aff1Al[0  , 0] := 1.00000E+01; aff1Al[0  , 1] := -9.84199E+00;
aff1Al[1  , 0] := 1.99800E+01; aff1Al[1  , 1] := -1.00077E+01;
aff1Al[2  , 0] := 2.99600E+01; aff1Al[2  , 1] := -1.02348E+01;
aff1Al[3  , 0] := 3.99400E+01; aff1Al[3  , 1] := -1.05422E+01;
aff1Al[4  , 0] := 4.99200E+01; aff1Al[4  , 1] := -1.10354E+01;
aff1Al[5  , 0] := 5.99000E+01; aff1Al[5  , 1] := -1.19198E+01;
aff1Al[6  , 0] := 6.98800E+01; aff1Al[6  , 1] := -1.41453E+01;
aff1Al[7  , 0] := 7.98600E+01; aff1Al[7  , 1] := -1.44478E+01;
aff1Al[8  , 0] := 8.98400E+01; aff1Al[8  , 1] := -1.31089E+01;
aff1Al[9  , 0] := 9.98200E+01; aff1Al[9  , 1] := -1.16796E+01;
aff1Al[10 , 0] := 1.09800E+02; aff1Al[10 , 1] := -1.03556E+01;
aff1Al[11 , 0] := 1.19780E+02; aff1Al[11 , 1] := -9.31746E+00;
aff1Al[12 , 0] := 1.29760E+02; aff1Al[12 , 1] := -7.63743E+00;
aff1Al[13 , 0] := 1.39740E+02; aff1Al[13 , 1] := -6.42389E+00;
aff1Al[14 , 0] := 1.49720E+02; aff1Al[14 , 1] := -5.44289E+00;
aff1Al[15 , 0] := 1.59700E+02; aff1Al[15 , 1] := -4.64208E+00;
aff1Al[16 , 0] := 1.69680E+02; aff1Al[16 , 1] := -3.98698E+00;
aff1Al[17 , 0] := 1.79660E+02; aff1Al[17 , 1] := -3.45000E+00;
aff1Al[18 , 0] := 1.89640E+02; aff1Al[18 , 1] := -3.00860E+00;
aff1Al[19 , 0] := 1.99620E+02; aff1Al[19 , 1] := -2.64455E+00;
aff1Al[20 , 0] := 2.09600E+02; aff1Al[20 , 1] := -2.34326E+00;
aff1Al[21 , 0] := 2.19580E+02; aff1Al[21 , 1] := -2.09321E+00;
aff1Al[22 , 0] := 2.29560E+02; aff1Al[22 , 1] := -1.88468E+00;
aff1Al[23 , 0] := 2.39540E+02; aff1Al[23 , 1] := -1.71030E+00;
aff1Al[24 , 0] := 2.49520E+02; aff1Al[24 , 1] := -1.56408E+00;
aff1Al[25 , 0] := 2.59500E+02; aff1Al[25 , 1] := -1.44116E+00;
aff1Al[26 , 0] := 2.69480E+02; aff1Al[26 , 1] := -1.33759E+00;
aff1Al[27 , 0] := 2.79460E+02; aff1Al[27 , 1] := -1.25018E+00;
aff1Al[28 , 0] := 2.89440E+02; aff1Al[28 , 1] := -1.17627E+00;
aff1Al[29 , 0] := 2.99420E+02; aff1Al[29 , 1] := -1.11369E+00;
aff1Al[30 , 0] := 3.09400E+02; aff1Al[30 , 1] := -1.06082E+00;
aff1Al[31 , 0] := 3.19380E+02; aff1Al[31 , 1] := -1.01635E+00;
aff1Al[32 , 0] := 3.29360E+02; aff1Al[32 , 1] := -9.79160E-01;
aff1Al[33 , 0] := 3.39340E+02; aff1Al[33 , 1] := -9.48230E-01;
aff1Al[34 , 0] := 3.49320E+02; aff1Al[34 , 1] := -9.22697E-01;
aff1Al[35 , 0] := 3.59300E+02; aff1Al[35 , 1] := -9.02016E-01;
aff1Al[36 , 0] := 3.69280E+02; aff1Al[36 , 1] := -8.85231E-01;
aff1Al[37 , 0] := 3.79260E+02; aff1Al[37 , 1] := -8.71960E-01;
aff1Al[38 , 0] := 3.89240E+02; aff1Al[38 , 1] := -8.61750E-01;
aff1Al[39 , 0] := 3.99220E+02; aff1Al[39 , 1] := -8.54204E-01;
aff1Al[40 , 0] := 4.09200E+02; aff1Al[40 , 1] := -8.48983E-01;
aff1Al[41 , 0] := 4.19180E+02; aff1Al[41 , 1] := -8.45791E-01;
aff1Al[42 , 0] := 4.29160E+02; aff1Al[42 , 1] := -8.44376E-01;
aff1Al[43 , 0] := 4.39140E+02; aff1Al[43 , 1] := -8.44514E-01;
aff1Al[44 , 0] := 4.49120E+02; aff1Al[44 , 1] := -8.46014E-01;
aff1Al[45 , 0] := 4.59100E+02; aff1Al[45 , 1] := -8.48707E-01;
aff1Al[46 , 0] := 4.69080E+02; aff1Al[46 , 1] := -8.52446E-01;
aff1Al[47 , 0] := 4.79060E+02; aff1Al[47 , 1] := -8.57102E-01;
aff1Al[48 , 0] := 4.89040E+02; aff1Al[48 , 1] := -8.62576E-01;
aff1Al[49 , 0] := 4.99020E+02; aff1Al[49 , 1] := -8.68781E-01;
aff1Al[50 , 0] := 5.09000E+02; aff1Al[50 , 1] := -8.75639E-01;
aff1Al[51 , 0] := 5.18980E+02; aff1Al[51 , 1] := -8.83079E-01;
aff1Al[52 , 0] := 5.28960E+02; aff1Al[52 , 1] := -8.91040E-01;
aff1Al[53 , 0] := 5.38940E+02; aff1Al[53 , 1] := -8.99464E-01;
aff1Al[54 , 0] := 5.48920E+02; aff1Al[54 , 1] := -9.08301E-01;
aff1Al[55 , 0] := 5.58900E+02; aff1Al[55 , 1] := -9.17508E-01;
aff1Al[56 , 0] := 5.68880E+02; aff1Al[56 , 1] := -9.27045E-01;
aff1Al[57 , 0] := 5.78860E+02; aff1Al[57 , 1] := -9.36877E-01;
aff1Al[58 , 0] := 5.88840E+02; aff1Al[58 , 1] := -9.46974E-01;
aff1Al[59 , 0] := 5.98820E+02; aff1Al[59 , 1] := -9.57307E-01;
aff1Al[60 , 0] := 6.08800E+02; aff1Al[60 , 1] := -9.67854E-01;
aff1Al[61 , 0] := 6.18780E+02; aff1Al[61 , 1] := -9.78593E-01;
aff1Al[62 , 0] := 6.28760E+02; aff1Al[62 , 1] := -9.89506E-01;
aff1Al[63 , 0] := 6.38740E+02; aff1Al[63 , 1] := -1.00058E+00;
aff1Al[64 , 0] := 6.48720E+02; aff1Al[64 , 1] := -1.01179E+00;
aff1Al[65 , 0] := 6.58700E+02; aff1Al[65 , 1] := -1.02313E+00;
aff1Al[66 , 0] := 6.68680E+02; aff1Al[66 , 1] := -1.03460E+00;
aff1Al[67 , 0] := 6.78660E+02; aff1Al[67 , 1] := -1.04617E+00;
aff1Al[68 , 0] := 6.88640E+02; aff1Al[68 , 1] := -1.05785E+00;
aff1Al[69 , 0] := 6.98620E+02; aff1Al[69 , 1] := -1.06963E+00;
aff1Al[70 , 0] := 7.08600E+02; aff1Al[70 , 1] := -1.08150E+00;
aff1Al[71 , 0] := 7.18580E+02; aff1Al[71 , 1] := -1.09346E+00;
aff1Al[72 , 0] := 7.28560E+02; aff1Al[72 , 1] := -1.10551E+00;
aff1Al[73 , 0] := 7.38540E+02; aff1Al[73 , 1] := -1.11763E+00;
aff1Al[74 , 0] := 7.48520E+02; aff1Al[74 , 1] := -1.12984E+00;
aff1Al[75 , 0] := 7.58500E+02; aff1Al[75 , 1] := -1.14213E+00;
aff1Al[76 , 0] := 7.68480E+02; aff1Al[76 , 1] := -1.15450E+00;
aff1Al[77 , 0] := 7.78460E+02; aff1Al[77 , 1] := -1.16695E+00;
aff1Al[78 , 0] := 7.88440E+02; aff1Al[78 , 1] := -1.17949E+00;
aff1Al[79 , 0] := 7.98420E+02; aff1Al[79 , 1] := -1.19211E+00;
aff1Al[80 , 0] := 8.08400E+02; aff1Al[80 , 1] := -1.20481E+00;
aff1Al[81 , 0] := 8.18380E+02; aff1Al[81 , 1] := -1.21760E+00;
aff1Al[82 , 0] := 8.28360E+02; aff1Al[82 , 1] := -1.23049E+00;
aff1Al[83 , 0] := 8.38340E+02; aff1Al[83 , 1] := -1.24347E+00;
aff1Al[84 , 0] := 8.48320E+02; aff1Al[84 , 1] := -1.25655E+00;
aff1Al[85 , 0] := 8.58300E+02; aff1Al[85 , 1] := -1.26974E+00;
aff1Al[86 , 0] := 8.68280E+02; aff1Al[86 , 1] := -1.28303E+00;
aff1Al[87 , 0] := 8.78260E+02; aff1Al[87 , 1] := -1.29644E+00;
aff1Al[88 , 0] := 8.88240E+02; aff1Al[88 , 1] := -1.30997E+00;
aff1Al[89 , 0] := 8.98220E+02; aff1Al[89 , 1] := -1.32363E+00;
aff1Al[90 , 0] := 9.08200E+02; aff1Al[90 , 1] := -1.33742E+00;
aff1Al[91 , 0] := 9.18180E+02; aff1Al[91 , 1] := -1.35136E+00;
aff1Al[92 , 0] := 9.28160E+02; aff1Al[92 , 1] := -1.36544E+00;
aff1Al[93 , 0] := 9.38140E+02; aff1Al[93 , 1] := -1.37968E+00;
aff1Al[94 , 0] := 9.48120E+02; aff1Al[94 , 1] := -1.39408E+00;
aff1Al[95 , 0] := 9.58100E+02; aff1Al[95 , 1] := -1.40865E+00;
aff1Al[96 , 0] := 9.68080E+02; aff1Al[96 , 1] := -1.42341E+00;
aff1Al[97 , 0] := 9.78060E+02; aff1Al[97 , 1] := -1.43836E+00;
aff1Al[98 , 0] := 9.88040E+02; aff1Al[98 , 1] := -1.45353E+00;
aff1Al[99 , 0] := 9.98020E+02; aff1Al[99 , 1] := -1.46877E+00;
aff1Al[100, 0] := 1.00800E+03; aff1Al[100, 1] := -1.47677E+00;
aff1Al[101, 0] := 1.01798E+03; aff1Al[101, 1] := -1.49037E+00;
aff1Al[102, 0] := 1.02796E+03; aff1Al[102, 1] := -1.50547E+00;
aff1Al[103, 0] := 1.03794E+03; aff1Al[103, 1] := -1.52135E+00;
aff1Al[104, 0] := 1.04792E+03; aff1Al[104, 1] := -1.53779E+00;
aff1Al[105, 0] := 1.05790E+03; aff1Al[105, 1] := -1.55471E+00;
aff1Al[106, 0] := 1.06788E+03; aff1Al[106, 1] := -1.57209E+00;
aff1Al[107, 0] := 1.07786E+03; aff1Al[107, 1] := -1.58990E+00;
aff1Al[108, 0] := 1.08784E+03; aff1Al[108, 1] := -1.60814E+00;
aff1Al[109, 0] := 1.09782E+03; aff1Al[109, 1] := -1.62683E+00;
aff1Al[110, 0] := 1.10780E+03; aff1Al[110, 1] := -1.64597E+00;
aff1Al[111, 0] := 1.11778E+03; aff1Al[111, 1] := -1.66557E+00;
aff1Al[112, 0] := 1.12776E+03; aff1Al[112, 1] := -1.68565E+00;
aff1Al[113, 0] := 1.13774E+03; aff1Al[113, 1] := -1.70624E+00;
aff1Al[114, 0] := 1.14772E+03; aff1Al[114, 1] := -1.72735E+00;
aff1Al[115, 0] := 1.15770E+03; aff1Al[115, 1] := -1.74901E+00;
aff1Al[116, 0] := 1.16768E+03; aff1Al[116, 1] := -1.77126E+00;
aff1Al[117, 0] := 1.17766E+03; aff1Al[117, 1] := -1.79411E+00;
aff1Al[118, 0] := 1.18764E+03; aff1Al[118, 1] := -1.81762E+00;
aff1Al[119, 0] := 1.19762E+03; aff1Al[119, 1] := -1.84181E+00;
aff1Al[120, 0] := 1.20760E+03; aff1Al[120, 1] := -1.86674E+00;
aff1Al[121, 0] := 1.21758E+03; aff1Al[121, 1] := -1.89244E+00;
aff1Al[122, 0] := 1.22756E+03; aff1Al[122, 1] := -1.91897E+00;
aff1Al[123, 0] := 1.23754E+03; aff1Al[123, 1] := -1.94639E+00;
aff1Al[124, 0] := 1.24752E+03; aff1Al[124, 1] := -1.97475E+00;
aff1Al[125, 0] := 1.25750E+03; aff1Al[125, 1] := -2.00414E+00;
aff1Al[126, 0] := 1.26748E+03; aff1Al[126, 1] := -2.03461E+00;
aff1Al[127, 0] := 1.27746E+03; aff1Al[127, 1] := -2.06626E+00;
aff1Al[128, 0] := 1.28744E+03; aff1Al[128, 1] := -2.09918E+00;
aff1Al[129, 0] := 1.29742E+03; aff1Al[129, 1] := -2.13348E+00;
aff1Al[130, 0] := 1.30740E+03; aff1Al[130, 1] := -2.16927E+00;
aff1Al[131, 0] := 1.31738E+03; aff1Al[131, 1] := -2.20668E+00;
aff1Al[132, 0] := 1.32736E+03; aff1Al[132, 1] := -2.24586E+00;
aff1Al[133, 0] := 1.33734E+03; aff1Al[133, 1] := -2.28699E+00;
aff1Al[134, 0] := 1.34732E+03; aff1Al[134, 1] := -2.33024E+00;
aff1Al[135, 0] := 1.35730E+03; aff1Al[135, 1] := -2.37585E+00;
aff1Al[136, 0] := 1.36728E+03; aff1Al[136, 1] := -2.42407E+00;
aff1Al[137, 0] := 1.37726E+03; aff1Al[137, 1] := -2.47520E+00;
aff1Al[138, 0] := 1.38724E+03; aff1Al[138, 1] := -2.52958E+00;
aff1Al[139, 0] := 1.39722E+03; aff1Al[139, 1] := -2.58764E+00;
aff1Al[140, 0] := 1.40720E+03; aff1Al[140, 1] := -2.64987E+00;
aff1Al[141, 0] := 1.41718E+03; aff1Al[141, 1] := -2.71687E+00;
aff1Al[142, 0] := 1.42716E+03; aff1Al[142, 1] := -2.78934E+00;
aff1Al[143, 0] := 1.43714E+03; aff1Al[143, 1] := -2.86819E+00;
aff1Al[144, 0] := 1.44712E+03; aff1Al[144, 1] := -2.95455E+00;
aff1Al[145, 0] := 1.45710E+03; aff1Al[145, 1] := -3.04985E+00;
aff1Al[146, 0] := 1.46708E+03; aff1Al[146, 1] := -3.15601E+00;
aff1Al[147, 0] := 1.47706E+03; aff1Al[147, 1] := -3.27556E+00;
aff1Al[148, 0] := 1.48704E+03; aff1Al[148, 1] := -3.41203E+00;
aff1Al[149, 0] := 1.49702E+03; aff1Al[149, 1] := -3.57073E+00;
aff1Al[150, 0] := 1.50700E+03; aff1Al[150, 1] := -3.75998E+00;
aff1Al[151, 0] := 1.51698E+03; aff1Al[151, 1] := -3.99072E+00;
aff1Al[152, 0] := 1.52696E+03; aff1Al[152, 1] := -4.28999E+00;
aff1Al[153, 0] := 1.53694E+03; aff1Al[153, 1] := -4.69289E+00;
aff1Al[154, 0] := 1.54692E+03; aff1Al[154, 1] := -5.36933E+00;
aff1Al[155, 0] := 1.55690E+03; aff1Al[155, 1] := -7.18317E+00;
aff1Al[156, 0] := 1.56688E+03; aff1Al[156, 1] := -6.04049E+00;
aff1Al[157, 0] := 1.57686E+03; aff1Al[157, 1] := -4.98882E+00;
aff1Al[158, 0] := 1.58684E+03; aff1Al[158, 1] := -4.41253E+00;
aff1Al[159, 0] := 1.59682E+03; aff1Al[159, 1] := -4.02524E+00;
aff1Al[160, 0] := 1.60680E+03; aff1Al[160, 1] := -3.71526E+00;
aff1Al[161, 0] := 1.61678E+03; aff1Al[161, 1] := -3.45829E+00;
aff1Al[162, 0] := 1.62676E+03; aff1Al[162, 1] := -3.23561E+00;
aff1Al[163, 0] := 1.63674E+03; aff1Al[163, 1] := -3.03403E+00;
aff1Al[164, 0] := 1.64672E+03; aff1Al[164, 1] := -2.85340E+00;
aff1Al[165, 0] := 1.65670E+03; aff1Al[165, 1] := -2.69189E+00;
aff1Al[166, 0] := 1.66668E+03; aff1Al[166, 1] := -2.54596E+00;
aff1Al[167, 0] := 1.67666E+03; aff1Al[167, 1] := -2.41278E+00;
aff1Al[168, 0] := 1.68664E+03; aff1Al[168, 1] := -2.28993E+00;
aff1Al[169, 0] := 1.69662E+03; aff1Al[169, 1] := -2.17603E+00;
aff1Al[170, 0] := 1.70660E+03; aff1Al[170, 1] := -2.06993E+00;
aff1Al[171, 0] := 1.71658E+03; aff1Al[171, 1] := -1.97068E+00;
aff1Al[172, 0] := 1.72656E+03; aff1Al[172, 1] := -1.87755E+00;
aff1Al[173, 0] := 1.73654E+03; aff1Al[173, 1] := -1.78991E+00;
aff1Al[174, 0] := 1.74652E+03; aff1Al[174, 1] := -1.70725E+00;
aff1Al[175, 0] := 1.75650E+03; aff1Al[175, 1] := -1.62914E+00;
aff1Al[176, 0] := 1.76648E+03; aff1Al[176, 1] := -1.55520E+00;
aff1Al[177, 0] := 1.77646E+03; aff1Al[177, 1] := -1.48511E+00;
aff1Al[178, 0] := 1.78644E+03; aff1Al[178, 1] := -1.41857E+00;
aff1Al[179, 0] := 1.79642E+03; aff1Al[179, 1] := -1.35535E+00;
aff1Al[180, 0] := 1.80640E+03; aff1Al[180, 1] := -1.29521E+00;
aff1Al[181, 0] := 1.81638E+03; aff1Al[181, 1] := -1.23796E+00;
aff1Al[182, 0] := 1.82636E+03; aff1Al[182, 1] := -1.18341E+00;
aff1Al[183, 0] := 1.83634E+03; aff1Al[183, 1] := -1.13142E+00;
aff1Al[184, 0] := 1.84632E+03; aff1Al[184, 1] := -1.08181E+00;
aff1Al[185, 0] := 1.85630E+03; aff1Al[185, 1] := -1.03447E+00;
aff1Al[186, 0] := 1.86628E+03; aff1Al[186, 1] := -9.89263E-01;
aff1Al[187, 0] := 1.87626E+03; aff1Al[187, 1] := -9.46076E-01;
aff1Al[188, 0] := 1.88624E+03; aff1Al[188, 1] := -9.04806E-01;
aff1Al[189, 0] := 1.89622E+03; aff1Al[189, 1] := -8.65352E-01;
aff1Al[190, 0] := 1.90620E+03; aff1Al[190, 1] := -8.27626E-01;
aff1Al[191, 0] := 1.91618E+03; aff1Al[191, 1] := -7.91542E-01;
aff1Al[192, 0] := 1.92616E+03; aff1Al[192, 1] := -7.57024E-01;
aff1Al[193, 0] := 1.93614E+03; aff1Al[193, 1] := -7.23998E-01;
aff1Al[194, 0] := 1.94612E+03; aff1Al[194, 1] := -6.92399E-01;
aff1Al[195, 0] := 1.95610E+03; aff1Al[195, 1] := -6.62165E-01;
aff1Al[196, 0] := 1.96608E+03; aff1Al[196, 1] := -6.33242E-01;
aff1Al[197, 0] := 1.97606E+03; aff1Al[197, 1] := -6.05580E-01;
aff1Al[198, 0] := 1.98604E+03; aff1Al[198, 1] := -5.79132E-01;
aff1Al[199, 0] := 1.99602E+03; aff1Al[199, 1] := -5.53864E-01;
aff1Al[200, 0] := 2.00600E+03; aff1Al[200, 1] := -5.29790E-01;
aff1Al[201, 0] := 2.01598E+03; aff1Al[201, 1] := -5.06864E-01;
aff1Al[202, 0] := 2.02596E+03; aff1Al[202, 1] := -4.84983E-01;
aff1Al[203, 0] := 2.03594E+03; aff1Al[203, 1] := -4.63991E-01;
aff1Al[204, 0] := 2.04592E+03; aff1Al[204, 1] := -4.43605E-01;
aff1Al[205, 0] := 2.05590E+03; aff1Al[205, 1] := -4.23670E-01;
aff1Al[206, 0] := 2.06588E+03; aff1Al[206, 1] := -4.04256E-01;
aff1Al[207, 0] := 2.07586E+03; aff1Al[207, 1] := -3.85410E-01;
aff1Al[208, 0] := 2.08584E+03; aff1Al[208, 1] := -3.67104E-01;
aff1Al[209, 0] := 2.09582E+03; aff1Al[209, 1] := -3.49316E-01;
aff1Al[210, 0] := 2.10580E+03; aff1Al[210, 1] := -3.32036E-01;
aff1Al[211, 0] := 2.11578E+03; aff1Al[211, 1] := -3.15248E-01;
aff1Al[212, 0] := 2.12576E+03; aff1Al[212, 1] := -2.98937E-01;
aff1Al[213, 0] := 2.13574E+03; aff1Al[213, 1] := -2.83087E-01;
aff1Al[214, 0] := 2.14572E+03; aff1Al[214, 1] := -2.67681E-01;
aff1Al[215, 0] := 2.15570E+03; aff1Al[215, 1] := -2.52704E-01;
aff1Al[216, 0] := 2.16568E+03; aff1Al[216, 1] := -2.38139E-01;
aff1Al[217, 0] := 2.17566E+03; aff1Al[217, 1] := -2.23973E-01;
aff1Al[218, 0] := 2.18564E+03; aff1Al[218, 1] := -2.10191E-01;
aff1Al[219, 0] := 2.19562E+03; aff1Al[219, 1] := -1.96778E-01;
aff1Al[220, 0] := 2.20560E+03; aff1Al[220, 1] := -1.83722E-01;
aff1Al[221, 0] := 2.21558E+03; aff1Al[221, 1] := -1.71010E-01;
aff1Al[222, 0] := 2.22556E+03; aff1Al[222, 1] := -1.58630E-01;
aff1Al[223, 0] := 2.23554E+03; aff1Al[223, 1] := -1.46573E-01;
aff1Al[224, 0] := 2.24552E+03; aff1Al[224, 1] := -1.34830E-01;
aff1Al[225, 0] := 2.25550E+03; aff1Al[225, 1] := -1.23388E-01;
aff1Al[226, 0] := 2.26548E+03; aff1Al[226, 1] := -1.12239E-01;
aff1Al[227, 0] := 2.27546E+03; aff1Al[227, 1] := -1.01370E-01;
aff1Al[228, 0] := 2.28544E+03; aff1Al[228, 1] := -9.07737E-02;
aff1Al[229, 0] := 2.29542E+03; aff1Al[229, 1] := -8.04398E-02;
aff1Al[230, 0] := 2.30540E+03; aff1Al[230, 1] := -7.03599E-02;
aff1Al[231, 0] := 2.31538E+03; aff1Al[231, 1] := -6.05256E-02;
aff1Al[232, 0] := 2.32536E+03; aff1Al[232, 1] := -5.09289E-02;
aff1Al[233, 0] := 2.33534E+03; aff1Al[233, 1] := -4.15622E-02;
aff1Al[234, 0] := 2.34532E+03; aff1Al[234, 1] := -3.24183E-02;
aff1Al[235, 0] := 2.35530E+03; aff1Al[235, 1] := -2.34900E-02;
aff1Al[236, 0] := 2.36528E+03; aff1Al[236, 1] := -1.47706E-02;
aff1Al[237, 0] := 2.37526E+03; aff1Al[237, 1] := -6.25378E-03;
aff1Al[238, 0] := 2.38524E+03; aff1Al[238, 1] := 2.06666E-03;
aff1Al[239, 0] := 2.39522E+03; aff1Al[239, 1] := 1.01966E-02;
aff1Al[240, 0] := 2.40520E+03; aff1Al[240, 1] := 1.81418E-02;
aff1Al[241, 0] := 2.41518E+03; aff1Al[241, 1] := 2.59075E-02;
aff1Al[242, 0] := 2.42516E+03; aff1Al[242, 1] := 3.34991E-02;
aff1Al[243, 0] := 2.43514E+03; aff1Al[243, 1] := 4.09215E-02;
aff1Al[244, 0] := 2.44512E+03; aff1Al[244, 1] := 4.81795E-02;
aff1Al[245, 0] := 2.45510E+03; aff1Al[245, 1] := 5.52777E-02;
aff1Al[246, 0] := 2.46508E+03; aff1Al[246, 1] := 6.22206E-02;
aff1Al[247, 0] := 2.47506E+03; aff1Al[247, 1] := 6.90126E-02;
aff1Al[248, 0] := 2.48504E+03; aff1Al[248, 1] := 7.56575E-02;
aff1Al[249, 0] := 2.49502E+03; aff1Al[249, 1] := 8.21595E-02;
aff1Al[250, 0] := 2.50500E+03; aff1Al[250, 1] := 8.85222E-02;
aff1Al[251, 0] := 2.51498E+03; aff1Al[251, 1] := 9.47495E-02;
aff1Al[252, 0] := 2.52496E+03; aff1Al[252, 1] := 1.00845E-01;
aff1Al[253, 0] := 2.53494E+03; aff1Al[253, 1] := 1.06812E-01;
aff1Al[254, 0] := 2.54492E+03; aff1Al[254, 1] := 1.12653E-01;
aff1Al[255, 0] := 2.55490E+03; aff1Al[255, 1] := 1.18373E-01;
aff1Al[256, 0] := 2.56488E+03; aff1Al[256, 1] := 1.23973E-01;
aff1Al[257, 0] := 2.57486E+03; aff1Al[257, 1] := 1.29458E-01;
aff1Al[258, 0] := 2.58484E+03; aff1Al[258, 1] := 1.34829E-01;
aff1Al[259, 0] := 2.59482E+03; aff1Al[259, 1] := 1.40090E-01;
aff1Al[260, 0] := 2.60480E+03; aff1Al[260, 1] := 1.45244E-01;
aff1Al[261, 0] := 2.61478E+03; aff1Al[261, 1] := 1.50292E-01;
aff1Al[262, 0] := 2.62476E+03; aff1Al[262, 1] := 1.55239E-01;
aff1Al[263, 0] := 2.63474E+03; aff1Al[263, 1] := 1.60086E-01;
aff1Al[264, 0] := 2.64472E+03; aff1Al[264, 1] := 1.64833E-01;
aff1Al[265, 0] := 2.65470E+03; aff1Al[265, 1] := 1.69484E-01;
aff1Al[266, 0] := 2.66468E+03; aff1Al[266, 1] := 1.74040E-01;
aff1Al[267, 0] := 2.67466E+03; aff1Al[267, 1] := 1.78507E-01;
aff1Al[268, 0] := 2.68464E+03; aff1Al[268, 1] := 1.82888E-01;
aff1Al[269, 0] := 2.69462E+03; aff1Al[269, 1] := 1.87183E-01;
aff1Al[270, 0] := 2.70460E+03; aff1Al[270, 1] := 1.91394E-01;
aff1Al[271, 0] := 2.71458E+03; aff1Al[271, 1] := 1.95522E-01;
aff1Al[272, 0] := 2.72456E+03; aff1Al[272, 1] := 1.99569E-01;
aff1Al[273, 0] := 2.73454E+03; aff1Al[273, 1] := 2.03537E-01;
aff1Al[274, 0] := 2.74452E+03; aff1Al[274, 1] := 2.07429E-01;
aff1Al[275, 0] := 2.75450E+03; aff1Al[275, 1] := 2.11246E-01;
aff1Al[276, 0] := 2.76448E+03; aff1Al[276, 1] := 2.14990E-01;
aff1Al[277, 0] := 2.77446E+03; aff1Al[277, 1] := 2.18663E-01;
aff1Al[278, 0] := 2.78444E+03; aff1Al[278, 1] := 2.22266E-01;
aff1Al[279, 0] := 2.79442E+03; aff1Al[279, 1] := 2.25801E-01;
aff1Al[280, 0] := 2.80440E+03; aff1Al[280, 1] := 2.29270E-01;
aff1Al[281, 0] := 2.81438E+03; aff1Al[281, 1] := 2.32675E-01;
aff1Al[282, 0] := 2.82436E+03; aff1Al[282, 1] := 2.36016E-01;
aff1Al[283, 0] := 2.83434E+03; aff1Al[283, 1] := 2.39297E-01;
aff1Al[284, 0] := 2.84432E+03; aff1Al[284, 1] := 2.42518E-01;
aff1Al[285, 0] := 2.85430E+03; aff1Al[285, 1] := 2.45681E-01;
aff1Al[286, 0] := 2.86428E+03; aff1Al[286, 1] := 2.48789E-01;
aff1Al[287, 0] := 2.87426E+03; aff1Al[287, 1] := 2.51841E-01;
aff1Al[288, 0] := 2.88424E+03; aff1Al[288, 1] := 2.54841E-01;
aff1Al[289, 0] := 2.89422E+03; aff1Al[289, 1] := 2.57789E-01;
aff1Al[290, 0] := 2.90420E+03; aff1Al[290, 1] := 2.60688E-01;
aff1Al[291, 0] := 2.91418E+03; aff1Al[291, 1] := 2.63540E-01;
aff1Al[292, 0] := 2.92416E+03; aff1Al[292, 1] := 2.66349E-01;
aff1Al[293, 0] := 2.93414E+03; aff1Al[293, 1] := 2.69138E-01;
aff1Al[294, 0] := 2.94412E+03; aff1Al[294, 1] := 2.71862E-01;
aff1Al[295, 0] := 2.95410E+03; aff1Al[295, 1] := 2.74462E-01;
aff1Al[296, 0] := 2.96408E+03; aff1Al[296, 1] := 2.76910E-01;
aff1Al[297, 0] := 2.97406E+03; aff1Al[297, 1] := 2.79499E-01;
aff1Al[298, 0] := 2.98404E+03; aff1Al[298, 1] := 2.82539E-01;
aff1Al[299, 0] := 2.99402E+03; aff1Al[299, 1] := 2.86146E-01;
aff1Al[300, 0] := 3.00400E+03; aff1Al[300, 1] := 2.89853E-01;
aff1Al[301, 0] := 3.01398E+03; aff1Al[301, 1] := 2.93173E-01;
aff1Al[302, 0] := 3.02396E+03; aff1Al[302, 1] := 2.95852E-01;
aff1Al[303, 0] := 3.03394E+03; aff1Al[303, 1] := 2.98120E-01;
aff1Al[304, 0] := 3.04392E+03; aff1Al[304, 1] := 3.00329E-01;
aff1Al[305, 0] := 3.05390E+03; aff1Al[305, 1] := 3.02814E-01;
aff1Al[306, 0] := 3.06388E+03; aff1Al[306, 1] := 3.04933E-01;
aff1Al[307, 0] := 3.07386E+03; aff1Al[307, 1] := 3.05880E-01;
aff1Al[308, 0] := 3.08384E+03; aff1Al[308, 1] := 3.05153E-01;
aff1Al[309, 0] := 3.09382E+03; aff1Al[309, 1] := 3.06508E-01;
aff1Al[310, 0] := 3.10380E+03; aff1Al[310, 1] := 3.13763E-01;
aff1Al[311, 0] := 3.11378E+03; aff1Al[311, 1] := 3.29581E-01;
aff1Al[312, 0] := 3.12376E+03; aff1Al[312, 1] := 3.48098E-01;
aff1Al[313, 0] := 3.13374E+03; aff1Al[313, 1] := 3.63012E-01;
aff1Al[314, 0] := 3.14372E+03; aff1Al[314, 1] := 3.69087E-01;
aff1Al[315, 0] := 3.15370E+03; aff1Al[315, 1] := 3.69334E-01;
aff1Al[316, 0] := 3.16368E+03; aff1Al[316, 1] := 3.67698E-01;
aff1Al[317, 0] := 3.17366E+03; aff1Al[317, 1] := 3.67875E-01;
aff1Al[318, 0] := 3.18364E+03; aff1Al[318, 1] := 3.69502E-01;
aff1Al[319, 0] := 3.19362E+03; aff1Al[319, 1] := 3.71637E-01;
aff1Al[320, 0] := 3.20360E+03; aff1Al[320, 1] := 3.73286E-01;
aff1Al[321, 0] := 3.21358E+03; aff1Al[321, 1] := 3.74565E-01;
aff1Al[322, 0] := 3.22356E+03; aff1Al[322, 1] := 3.75687E-01;
aff1Al[323, 0] := 3.23354E+03; aff1Al[323, 1] := 3.76814E-01;
aff1Al[324, 0] := 3.24352E+03; aff1Al[324, 1] := 3.77939E-01;
aff1Al[325, 0] := 3.25350E+03; aff1Al[325, 1] := 3.79018E-01;
aff1Al[326, 0] := 3.26348E+03; aff1Al[326, 1] := 3.80052E-01;
aff1Al[327, 0] := 3.27346E+03; aff1Al[327, 1] := 3.81042E-01;
aff1Al[328, 0] := 3.28344E+03; aff1Al[328, 1] := 3.81991E-01;
aff1Al[329, 0] := 3.29342E+03; aff1Al[329, 1] := 3.82900E-01;
aff1Al[330, 0] := 3.30340E+03; aff1Al[330, 1] := 3.83769E-01;
aff1Al[331, 0] := 3.31338E+03; aff1Al[331, 1] := 3.84601E-01;
aff1Al[332, 0] := 3.32336E+03; aff1Al[332, 1] := 3.85396E-01;
aff1Al[333, 0] := 3.33334E+03; aff1Al[333, 1] := 3.86155E-01;
aff1Al[334, 0] := 3.34332E+03; aff1Al[334, 1] := 3.86880E-01;
aff1Al[335, 0] := 3.35330E+03; aff1Al[335, 1] := 3.87572E-01;
aff1Al[336, 0] := 3.36328E+03; aff1Al[336, 1] := 3.88231E-01;
aff1Al[337, 0] := 3.37326E+03; aff1Al[337, 1] := 3.88859E-01;
aff1Al[338, 0] := 3.38324E+03; aff1Al[338, 1] := 3.89456E-01;
aff1Al[339, 0] := 3.39322E+03; aff1Al[339, 1] := 3.90023E-01;
aff1Al[340, 0] := 3.40320E+03; aff1Al[340, 1] := 3.90562E-01;
aff1Al[341, 0] := 3.41318E+03; aff1Al[341, 1] := 3.91072E-01;
aff1Al[342, 0] := 3.42316E+03; aff1Al[342, 1] := 3.91555E-01;
aff1Al[343, 0] := 3.43314E+03; aff1Al[343, 1] := 3.92012E-01;
aff1Al[344, 0] := 3.44312E+03; aff1Al[344, 1] := 3.92443E-01;
aff1Al[345, 0] := 3.45310E+03; aff1Al[345, 1] := 3.92848E-01;
aff1Al[346, 0] := 3.46308E+03; aff1Al[346, 1] := 3.93229E-01;
aff1Al[347, 0] := 3.47306E+03; aff1Al[347, 1] := 3.93586E-01;
aff1Al[348, 0] := 3.48304E+03; aff1Al[348, 1] := 3.93920E-01;
aff1Al[349, 0] := 3.49302E+03; aff1Al[349, 1] := 3.94231E-01;
aff1Al[350, 0] := 3.50300E+03; aff1Al[350, 1] := 3.94520E-01;
aff1Al[351, 0] := 3.51298E+03; aff1Al[351, 1] := 3.94787E-01;
aff1Al[352, 0] := 3.52296E+03; aff1Al[352, 1] := 3.95033E-01;
aff1Al[353, 0] := 3.53294E+03; aff1Al[353, 1] := 3.95259E-01;
aff1Al[354, 0] := 3.54292E+03; aff1Al[354, 1] := 3.95465E-01;
aff1Al[355, 0] := 3.55290E+03; aff1Al[355, 1] := 3.95652E-01;
aff1Al[356, 0] := 3.56288E+03; aff1Al[356, 1] := 3.95819E-01;
aff1Al[357, 0] := 3.57286E+03; aff1Al[357, 1] := 3.95968E-01;
aff1Al[358, 0] := 3.58284E+03; aff1Al[358, 1] := 3.96099E-01;
aff1Al[359, 0] := 3.59282E+03; aff1Al[359, 1] := 3.96213E-01;
aff1Al[360, 0] := 3.60280E+03; aff1Al[360, 1] := 3.96309E-01;
aff1Al[361, 0] := 3.61278E+03; aff1Al[361, 1] := 3.96388E-01;
aff1Al[362, 0] := 3.62276E+03; aff1Al[362, 1] := 3.96451E-01;
aff1Al[363, 0] := 3.63274E+03; aff1Al[363, 1] := 3.96498E-01;
aff1Al[364, 0] := 3.64272E+03; aff1Al[364, 1] := 3.96529E-01;
aff1Al[365, 0] := 3.65270E+03; aff1Al[365, 1] := 3.96545E-01;
aff1Al[366, 0] := 3.66268E+03; aff1Al[366, 1] := 3.96547E-01;
aff1Al[367, 0] := 3.67266E+03; aff1Al[367, 1] := 3.96533E-01;
aff1Al[368, 0] := 3.68264E+03; aff1Al[368, 1] := 3.96506E-01;
aff1Al[369, 0] := 3.69262E+03; aff1Al[369, 1] := 3.96465E-01;
aff1Al[370, 0] := 3.70260E+03; aff1Al[370, 1] := 3.96410E-01;
aff1Al[371, 0] := 3.71258E+03; aff1Al[371, 1] := 3.96342E-01;
aff1Al[372, 0] := 3.72256E+03; aff1Al[372, 1] := 3.96261E-01;
aff1Al[373, 0] := 3.73254E+03; aff1Al[373, 1] := 3.96167E-01;
aff1Al[374, 0] := 3.74252E+03; aff1Al[374, 1] := 3.96062E-01;
aff1Al[375, 0] := 3.75250E+03; aff1Al[375, 1] := 3.95944E-01;
aff1Al[376, 0] := 3.76248E+03; aff1Al[376, 1] := 3.95814E-01;
aff1Al[377, 0] := 3.77246E+03; aff1Al[377, 1] := 3.95673E-01;
aff1Al[378, 0] := 3.78244E+03; aff1Al[378, 1] := 3.95521E-01;
aff1Al[379, 0] := 3.79242E+03; aff1Al[379, 1] := 3.95358E-01;
aff1Al[380, 0] := 3.80240E+03; aff1Al[380, 1] := 3.95184E-01;
aff1Al[381, 0] := 3.81238E+03; aff1Al[381, 1] := 3.95000E-01;
aff1Al[382, 0] := 3.82236E+03; aff1Al[382, 1] := 3.94806E-01;
aff1Al[383, 0] := 3.83234E+03; aff1Al[383, 1] := 3.94602E-01;
aff1Al[384, 0] := 3.84232E+03; aff1Al[384, 1] := 3.94388E-01;
aff1Al[385, 0] := 3.85230E+03; aff1Al[385, 1] := 3.94165E-01;
aff1Al[386, 0] := 3.86228E+03; aff1Al[386, 1] := 3.93932E-01;
aff1Al[387, 0] := 3.87226E+03; aff1Al[387, 1] := 3.93690E-01;
aff1Al[388, 0] := 3.88224E+03; aff1Al[388, 1] := 3.93440E-01;
aff1Al[389, 0] := 3.89222E+03; aff1Al[389, 1] := 3.93181E-01;
aff1Al[390, 0] := 3.90220E+03; aff1Al[390, 1] := 3.92913E-01;
aff1Al[391, 0] := 3.91218E+03; aff1Al[391, 1] := 3.92637E-01;
aff1Al[392, 0] := 3.92216E+03; aff1Al[392, 1] := 3.92353E-01;
aff1Al[393, 0] := 3.93214E+03; aff1Al[393, 1] := 3.92062E-01;
aff1Al[394, 0] := 3.94212E+03; aff1Al[394, 1] := 3.91762E-01;
aff1Al[395, 0] := 3.95210E+03; aff1Al[395, 1] := 3.91455E-01;
aff1Al[396, 0] := 3.96208E+03; aff1Al[396, 1] := 3.91141E-01;
aff1Al[397, 0] := 3.97206E+03; aff1Al[397, 1] := 3.90820E-01;
aff1Al[398, 0] := 3.98204E+03; aff1Al[398, 1] := 3.90491E-01;
aff1Al[399, 0] := 3.99202E+03; aff1Al[399, 1] := 3.90156E-01;
aff1Al[400, 0] := 4.00200E+03; aff1Al[400, 1] := 3.89814E-01;
aff1Al[401, 0] := 4.01198E+03; aff1Al[401, 1] := 3.89466E-01;
aff1Al[402, 0] := 4.02196E+03; aff1Al[402, 1] := 3.89111E-01;
aff1Al[403, 0] := 4.03194E+03; aff1Al[403, 1] := 3.88750E-01;
aff1Al[404, 0] := 4.04192E+03; aff1Al[404, 1] := 3.88384E-01;
aff1Al[405, 0] := 4.05190E+03; aff1Al[405, 1] := 3.88011E-01;
aff1Al[406, 0] := 4.06188E+03; aff1Al[406, 1] := 3.87632E-01;
aff1Al[407, 0] := 4.07186E+03; aff1Al[407, 1] := 3.87248E-01;
aff1Al[408, 0] := 4.08184E+03; aff1Al[408, 1] := 3.86859E-01;
aff1Al[409, 0] := 4.09182E+03; aff1Al[409, 1] := 3.86464E-01;
aff1Al[410, 0] := 4.10180E+03; aff1Al[410, 1] := 3.86064E-01;
aff1Al[411, 0] := 4.11178E+03; aff1Al[411, 1] := 3.85659E-01;
aff1Al[412, 0] := 4.12176E+03; aff1Al[412, 1] := 3.85249E-01;
aff1Al[413, 0] := 4.13174E+03; aff1Al[413, 1] := 3.84834E-01;
aff1Al[414, 0] := 4.14172E+03; aff1Al[414, 1] := 3.84413E-01;
aff1Al[415, 0] := 4.15170E+03; aff1Al[415, 1] := 3.83987E-01;
aff1Al[416, 0] := 4.16168E+03; aff1Al[416, 1] := 3.83557E-01;
aff1Al[417, 0] := 4.17166E+03; aff1Al[417, 1] := 3.83122E-01;
aff1Al[418, 0] := 4.18164E+03; aff1Al[418, 1] := 3.82683E-01;
aff1Al[419, 0] := 4.19162E+03; aff1Al[419, 1] := 3.82241E-01;
aff1Al[420, 0] := 4.20160E+03; aff1Al[420, 1] := 3.81795E-01;
aff1Al[421, 0] := 4.21158E+03; aff1Al[421, 1] := 3.81346E-01;
aff1Al[422, 0] := 4.22156E+03; aff1Al[422, 1] := 3.80893E-01;
aff1Al[423, 0] := 4.23154E+03; aff1Al[423, 1] := 3.80436E-01;
aff1Al[424, 0] := 4.24152E+03; aff1Al[424, 1] := 3.79975E-01;
aff1Al[425, 0] := 4.25150E+03; aff1Al[425, 1] := 3.79511E-01;
aff1Al[426, 0] := 4.26148E+03; aff1Al[426, 1] := 3.79043E-01;
aff1Al[427, 0] := 4.27146E+03; aff1Al[427, 1] := 3.78572E-01;
aff1Al[428, 0] := 4.28144E+03; aff1Al[428, 1] := 3.78097E-01;
aff1Al[429, 0] := 4.29142E+03; aff1Al[429, 1] := 3.77620E-01;
aff1Al[430, 0] := 4.30140E+03; aff1Al[430, 1] := 3.77139E-01;
aff1Al[431, 0] := 4.31138E+03; aff1Al[431, 1] := 3.76655E-01;
aff1Al[432, 0] := 4.32136E+03; aff1Al[432, 1] := 3.76168E-01;
aff1Al[433, 0] := 4.33134E+03; aff1Al[433, 1] := 3.75679E-01;
aff1Al[434, 0] := 4.34132E+03; aff1Al[434, 1] := 3.75187E-01;
aff1Al[435, 0] := 4.35130E+03; aff1Al[435, 1] := 3.74692E-01;
aff1Al[436, 0] := 4.36128E+03; aff1Al[436, 1] := 3.74194E-01;
aff1Al[437, 0] := 4.37126E+03; aff1Al[437, 1] := 3.73694E-01;
aff1Al[438, 0] := 4.38124E+03; aff1Al[438, 1] := 3.73191E-01;
aff1Al[439, 0] := 4.39122E+03; aff1Al[439, 1] := 3.72686E-01;
aff1Al[440, 0] := 4.40120E+03; aff1Al[440, 1] := 3.72179E-01;
aff1Al[441, 0] := 4.41118E+03; aff1Al[441, 1] := 3.71669E-01;
aff1Al[442, 0] := 4.42116E+03; aff1Al[442, 1] := 3.71157E-01;
aff1Al[443, 0] := 4.43114E+03; aff1Al[443, 1] := 3.70644E-01;
aff1Al[444, 0] := 4.44112E+03; aff1Al[444, 1] := 3.70128E-01;
aff1Al[445, 0] := 4.45110E+03; aff1Al[445, 1] := 3.69610E-01;
aff1Al[446, 0] := 4.46108E+03; aff1Al[446, 1] := 3.69090E-01;
aff1Al[447, 0] := 4.47106E+03; aff1Al[447, 1] := 3.68568E-01;
aff1Al[448, 0] := 4.48104E+03; aff1Al[448, 1] := 3.68045E-01;
aff1Al[449, 0] := 4.49102E+03; aff1Al[449, 1] := 3.67519E-01;
aff1Al[450, 0] := 4.50100E+03; aff1Al[450, 1] := 3.66992E-01;
aff1Al[451, 0] := 4.51098E+03; aff1Al[451, 1] := 3.66464E-01;
aff1Al[452, 0] := 4.52096E+03; aff1Al[452, 1] := 3.65934E-01;
aff1Al[453, 0] := 4.53094E+03; aff1Al[453, 1] := 3.65402E-01;
aff1Al[454, 0] := 4.54092E+03; aff1Al[454, 1] := 3.64869E-01;
aff1Al[455, 0] := 4.55090E+03; aff1Al[455, 1] := 3.64334E-01;
aff1Al[456, 0] := 4.56088E+03; aff1Al[456, 1] := 3.63798E-01;
aff1Al[457, 0] := 4.57086E+03; aff1Al[457, 1] := 3.63261E-01;
aff1Al[458, 0] := 4.58084E+03; aff1Al[458, 1] := 3.62723E-01;
aff1Al[459, 0] := 4.59082E+03; aff1Al[459, 1] := 3.62183E-01;
aff1Al[460, 0] := 4.60080E+03; aff1Al[460, 1] := 3.61642E-01;
aff1Al[461, 0] := 4.61078E+03; aff1Al[461, 1] := 3.61100E-01;
aff1Al[462, 0] := 4.62076E+03; aff1Al[462, 1] := 3.60557E-01;
aff1Al[463, 0] := 4.63074E+03; aff1Al[463, 1] := 3.60013E-01;
aff1Al[464, 0] := 4.64072E+03; aff1Al[464, 1] := 3.59468E-01;
aff1Al[465, 0] := 4.65070E+03; aff1Al[465, 1] := 3.58922E-01;
aff1Al[466, 0] := 4.66068E+03; aff1Al[466, 1] := 3.58375E-01;
aff1Al[467, 0] := 4.67066E+03; aff1Al[467, 1] := 3.57827E-01;
aff1Al[468, 0] := 4.68064E+03; aff1Al[468, 1] := 3.57278E-01;
aff1Al[469, 0] := 4.69062E+03; aff1Al[469, 1] := 3.56729E-01;
aff1Al[470, 0] := 4.70060E+03; aff1Al[470, 1] := 3.56179E-01;
aff1Al[471, 0] := 4.71058E+03; aff1Al[471, 1] := 3.55628E-01;
aff1Al[472, 0] := 4.72056E+03; aff1Al[472, 1] := 3.55076E-01;
aff1Al[473, 0] := 4.73054E+03; aff1Al[473, 1] := 3.54524E-01;
aff1Al[474, 0] := 4.74052E+03; aff1Al[474, 1] := 3.53972E-01;
aff1Al[475, 0] := 4.75050E+03; aff1Al[475, 1] := 3.53418E-01;
aff1Al[476, 0] := 4.76048E+03; aff1Al[476, 1] := 3.52865E-01;
aff1Al[477, 0] := 4.77046E+03; aff1Al[477, 1] := 3.52310E-01;
aff1Al[478, 0] := 4.78044E+03; aff1Al[478, 1] := 3.51756E-01;
aff1Al[479, 0] := 4.79042E+03; aff1Al[479, 1] := 3.51200E-01;
aff1Al[480, 0] := 4.80040E+03; aff1Al[480, 1] := 3.50645E-01;
aff1Al[481, 0] := 4.81038E+03; aff1Al[481, 1] := 3.50089E-01;
aff1Al[482, 0] := 4.82036E+03; aff1Al[482, 1] := 3.49533E-01;
aff1Al[483, 0] := 4.83034E+03; aff1Al[483, 1] := 3.48977E-01;
aff1Al[484, 0] := 4.84032E+03; aff1Al[484, 1] := 3.48420E-01;
aff1Al[485, 0] := 4.85030E+03; aff1Al[485, 1] := 3.47863E-01;
aff1Al[486, 0] := 4.86028E+03; aff1Al[486, 1] := 3.47306E-01;
aff1Al[487, 0] := 4.87026E+03; aff1Al[487, 1] := 3.46748E-01;
aff1Al[488, 0] := 4.88024E+03; aff1Al[488, 1] := 3.46191E-01;
aff1Al[489, 0] := 4.89022E+03; aff1Al[489, 1] := 3.45633E-01;
aff1Al[490, 0] := 4.90020E+03; aff1Al[490, 1] := 3.45076E-01;
aff1Al[491, 0] := 4.91018E+03; aff1Al[491, 1] := 3.44518E-01;
aff1Al[492, 0] := 4.92016E+03; aff1Al[492, 1] := 3.43960E-01;
aff1Al[493, 0] := 4.93014E+03; aff1Al[493, 1] := 3.43402E-01;
aff1Al[494, 0] := 4.94012E+03; aff1Al[494, 1] := 3.42845E-01;
aff1Al[495, 0] := 4.95010E+03; aff1Al[495, 1] := 3.42287E-01;
aff1Al[496, 0] := 4.96008E+03; aff1Al[496, 1] := 3.41729E-01;
aff1Al[497, 0] := 4.97006E+03; aff1Al[497, 1] := 3.41171E-01;
aff1Al[498, 0] := 4.98004E+03; aff1Al[498, 1] := 3.40614E-01;
aff1Al[499, 0] := 4.99002E+03; aff1Al[499, 1] := 3.40056E-01;
aff1Al[500, 0] := 5.00000E+03; aff1Al[500, 1] := 3.39499E-01;
aff1Al[501, 0] := 5.05000E+03; aff1Al[501, 1] := 3.36710E-01;
aff1Al[502, 0] := 5.10000E+03; aff1Al[502, 1] := 3.33928E-01;
aff1Al[503, 0] := 5.15000E+03; aff1Al[503, 1] := 3.31155E-01;
aff1Al[504, 0] := 5.20000E+03; aff1Al[504, 1] := 3.28393E-01;
aff1Al[505, 0] := 5.25000E+03; aff1Al[505, 1] := 3.25645E-01;
aff1Al[506, 0] := 5.30000E+03; aff1Al[506, 1] := 3.22911E-01;
aff1Al[507, 0] := 5.35000E+03; aff1Al[507, 1] := 3.20193E-01;
aff1Al[508, 0] := 5.40000E+03; aff1Al[508, 1] := 3.17493E-01;
aff1Al[509, 0] := 5.45000E+03; aff1Al[509, 1] := 3.14812E-01;
aff1Al[510, 0] := 5.50000E+03; aff1Al[510, 1] := 3.12152E-01;
aff1Al[511, 0] := 5.55000E+03; aff1Al[511, 1] := 3.09512E-01;
aff1Al[512, 0] := 5.60000E+03; aff1Al[512, 1] := 3.06895E-01;
aff1Al[513, 0] := 5.65000E+03; aff1Al[513, 1] := 3.04301E-01;
aff1Al[514, 0] := 5.70000E+03; aff1Al[514, 1] := 3.01730E-01;
aff1Al[515, 0] := 5.75000E+03; aff1Al[515, 1] := 2.99184E-01;
aff1Al[516, 0] := 5.80000E+03; aff1Al[516, 1] := 2.96662E-01;
aff1Al[517, 0] := 5.85000E+03; aff1Al[517, 1] := 2.94167E-01;
aff1Al[518, 0] := 5.90000E+03; aff1Al[518, 1] := 2.91697E-01;
aff1Al[519, 0] := 5.95000E+03; aff1Al[519, 1] := 2.89254E-01;
aff1Al[520, 0] := 6.00000E+03; aff1Al[520, 1] := 2.86838E-01;
aff1Al[521, 0] := 6.05000E+03; aff1Al[521, 1] := 2.84450E-01;
aff1Al[522, 0] := 6.10000E+03; aff1Al[522, 1] := 2.82089E-01;
aff1Al[523, 0] := 6.15000E+03; aff1Al[523, 1] := 2.79756E-01;
aff1Al[524, 0] := 6.20000E+03; aff1Al[524, 1] := 2.77451E-01;
aff1Al[525, 0] := 6.25000E+03; aff1Al[525, 1] := 2.75175E-01;
aff1Al[526, 0] := 6.30000E+03; aff1Al[526, 1] := 2.72928E-01;
aff1Al[527, 0] := 6.35000E+03; aff1Al[527, 1] := 2.70711E-01;
aff1Al[528, 0] := 6.40000E+03; aff1Al[528, 1] := 2.68523E-01;
aff1Al[529, 0] := 6.45000E+03; aff1Al[529, 1] := 2.66365E-01;
aff1Al[530, 0] := 6.50000E+03; aff1Al[530, 1] := 2.64237E-01;
aff1Al[531, 0] := 6.55000E+03; aff1Al[531, 1] := 2.62140E-01;
aff1Al[532, 0] := 6.60000E+03; aff1Al[532, 1] := 2.60075E-01;
aff1Al[533, 0] := 6.65000E+03; aff1Al[533, 1] := 2.58040E-01;
aff1Al[534, 0] := 6.70000E+03; aff1Al[534, 1] := 2.56039E-01;
aff1Al[535, 0] := 6.75000E+03; aff1Al[535, 1] := 2.54070E-01;
aff1Al[536, 0] := 6.80000E+03; aff1Al[536, 1] := 2.52130E-01;
aff1Al[537, 0] := 6.85000E+03; aff1Al[537, 1] := 2.50192E-01;
aff1Al[538, 0] := 6.90000E+03; aff1Al[538, 1] := 2.48253E-01;
aff1Al[539, 0] := 6.95000E+03; aff1Al[539, 1] := 2.46318E-01;
aff1Al[540, 0] := 7.00000E+03; aff1Al[540, 1] := 2.44389E-01;
aff1Al[541, 0] := 7.05000E+03; aff1Al[541, 1] := 2.42466E-01;
aff1Al[542, 0] := 7.10000E+03; aff1Al[542, 1] := 2.40553E-01;
aff1Al[543, 0] := 7.15000E+03; aff1Al[543, 1] := 2.38650E-01;
aff1Al[544, 0] := 7.20000E+03; aff1Al[544, 1] := 2.36757E-01;
aff1Al[545, 0] := 7.25000E+03; aff1Al[545, 1] := 2.34877E-01;
aff1Al[546, 0] := 7.30000E+03; aff1Al[546, 1] := 2.33010E-01;
aff1Al[547, 0] := 7.35000E+03; aff1Al[547, 1] := 2.31156E-01;
aff1Al[548, 0] := 7.40000E+03; aff1Al[548, 1] := 2.29316E-01;
aff1Al[549, 0] := 7.45000E+03; aff1Al[549, 1] := 2.27491E-01;
aff1Al[550, 0] := 7.50000E+03; aff1Al[550, 1] := 2.25681E-01;
aff1Al[551, 0] := 7.55000E+03; aff1Al[551, 1] := 2.23886E-01;
aff1Al[552, 0] := 7.60000E+03; aff1Al[552, 1] := 2.22107E-01;
aff1Al[553, 0] := 7.65000E+03; aff1Al[553, 1] := 2.20344E-01;
aff1Al[554, 0] := 7.70000E+03; aff1Al[554, 1] := 2.18596E-01;
aff1Al[555, 0] := 7.75000E+03; aff1Al[555, 1] := 2.16865E-01;
aff1Al[556, 0] := 7.80000E+03; aff1Al[556, 1] := 2.15150E-01;
aff1Al[557, 0] := 7.85000E+03; aff1Al[557, 1] := 2.13452E-01;
aff1Al[558, 0] := 7.90000E+03; aff1Al[558, 1] := 2.11770E-01;
aff1Al[559, 0] := 7.95000E+03; aff1Al[559, 1] := 2.10104E-01;
aff1Al[560, 0] := 8.00000E+03; aff1Al[560, 1] := 2.08455E-01;
aff1Al[561, 0] := 8.05000E+03; aff1Al[561, 1] := 2.06823E-01;
aff1Al[562, 0] := 8.10000E+03; aff1Al[562, 1] := 2.05207E-01;
aff1Al[563, 0] := 8.15000E+03; aff1Al[563, 1] := 2.03607E-01;
aff1Al[564, 0] := 8.20000E+03; aff1Al[564, 1] := 2.02024E-01;
aff1Al[565, 0] := 8.25000E+03; aff1Al[565, 1] := 2.00457E-01;
aff1Al[566, 0] := 8.30000E+03; aff1Al[566, 1] := 1.98907E-01;
aff1Al[567, 0] := 8.35000E+03; aff1Al[567, 1] := 1.97373E-01;
aff1Al[568, 0] := 8.40000E+03; aff1Al[568, 1] := 1.95855E-01;
aff1Al[569, 0] := 8.45000E+03; aff1Al[569, 1] := 1.94353E-01;
aff1Al[570, 0] := 8.50000E+03; aff1Al[570, 1] := 1.92868E-01;
aff1Al[571, 0] := 8.55000E+03; aff1Al[571, 1] := 1.91398E-01;
aff1Al[572, 0] := 8.60000E+03; aff1Al[572, 1] := 1.89944E-01;
aff1Al[573, 0] := 8.65000E+03; aff1Al[573, 1] := 1.88505E-01;
aff1Al[574, 0] := 8.70000E+03; aff1Al[574, 1] := 1.87083E-01;
aff1Al[575, 0] := 8.75000E+03; aff1Al[575, 1] := 1.85676E-01;
aff1Al[576, 0] := 8.80000E+03; aff1Al[576, 1] := 1.84285E-01;
aff1Al[577, 0] := 8.85000E+03; aff1Al[577, 1] := 1.82900E-01;
aff1Al[578, 0] := 8.90000E+03; aff1Al[578, 1] := 1.81562E-01;
aff1Al[579, 0] := 8.95000E+03; aff1Al[579, 1] := 1.80351E-01;
aff1Al[580, 0] := 9.00000E+03; aff1Al[580, 1] := 1.79197E-01;
aff1Al[581, 0] := 9.05000E+03; aff1Al[581, 1] := 1.78006E-01;
aff1Al[582, 0] := 9.10000E+03; aff1Al[582, 1] := 1.76795E-01;
aff1Al[583, 0] := 9.15000E+03; aff1Al[583, 1] := 1.75586E-01;
aff1Al[584, 0] := 9.20000E+03; aff1Al[584, 1] := 1.74375E-01;
aff1Al[585, 0] := 9.25000E+03; aff1Al[585, 1] := 1.73163E-01;
aff1Al[586, 0] := 9.30000E+03; aff1Al[586, 1] := 1.71951E-01;
aff1Al[587, 0] := 9.35000E+03; aff1Al[587, 1] := 1.70742E-01;
aff1Al[588, 0] := 9.40000E+03; aff1Al[588, 1] := 1.69535E-01;
aff1Al[589, 0] := 9.45000E+03; aff1Al[589, 1] := 1.68333E-01;
aff1Al[590, 0] := 9.50000E+03; aff1Al[590, 1] := 1.67136E-01;
aff1Al[591, 0] := 9.55000E+03; aff1Al[591, 1] := 1.65944E-01;
aff1Al[592, 0] := 9.60000E+03; aff1Al[592, 1] := 1.64758E-01;
aff1Al[593, 0] := 9.65000E+03; aff1Al[593, 1] := 1.63579E-01;
aff1Al[594, 0] := 9.70000E+03; aff1Al[594, 1] := 1.62407E-01;
aff1Al[595, 0] := 9.75000E+03; aff1Al[595, 1] := 1.61243E-01;
aff1Al[596, 0] := 9.80000E+03; aff1Al[596, 1] := 1.60086E-01;
aff1Al[597, 0] := 9.85000E+03; aff1Al[597, 1] := 1.58936E-01;
aff1Al[598, 0] := 9.90000E+03; aff1Al[598, 1] := 1.57795E-01;
aff1Al[599, 0] := 9.95000E+03; aff1Al[599, 1] := 1.56662E-01;
aff1Al[600, 0] := 1.00000E+04; aff1Al[600, 1] := 1.55537E-01;
aff1Al[601, 0] := 1.00500E+04; aff1Al[601, 1] := 1.54421E-01;
aff1Al[602, 0] := 1.01000E+04; aff1Al[602, 1] := 1.53314E-01;
aff1Al[603, 0] := 1.01500E+04; aff1Al[603, 1] := 1.52215E-01;
aff1Al[604, 0] := 1.02000E+04; aff1Al[604, 1] := 1.51124E-01;
aff1Al[605, 0] := 1.02500E+04; aff1Al[605, 1] := 1.50043E-01;
aff1Al[606, 0] := 1.03000E+04; aff1Al[606, 1] := 1.48970E-01;
aff1Al[607, 0] := 1.03500E+04; aff1Al[607, 1] := 1.47906E-01;
aff1Al[608, 0] := 1.04000E+04; aff1Al[608, 1] := 1.46850E-01;
aff1Al[609, 0] := 1.04500E+04; aff1Al[609, 1] := 1.45804E-01;
aff1Al[610, 0] := 1.05000E+04; aff1Al[610, 1] := 1.44766E-01;
aff1Al[611, 0] := 1.05500E+04; aff1Al[611, 1] := 1.43737E-01;
aff1Al[612, 0] := 1.06000E+04; aff1Al[612, 1] := 1.42717E-01;
aff1Al[613, 0] := 1.06500E+04; aff1Al[613, 1] := 1.41705E-01;
aff1Al[614, 0] := 1.07000E+04; aff1Al[614, 1] := 1.40702E-01;
aff1Al[615, 0] := 1.07500E+04; aff1Al[615, 1] := 1.39707E-01;
aff1Al[616, 0] := 1.08000E+04; aff1Al[616, 1] := 1.38721E-01;
aff1Al[617, 0] := 1.08500E+04; aff1Al[617, 1] := 1.37744E-01;
aff1Al[618, 0] := 1.09000E+04; aff1Al[618, 1] := 1.36775E-01;
aff1Al[619, 0] := 1.09500E+04; aff1Al[619, 1] := 1.35815E-01;
aff1Al[620, 0] := 1.10000E+04; aff1Al[620, 1] := 1.34862E-01;
aff1Al[621, 0] := 1.10500E+04; aff1Al[621, 1] := 1.33918E-01;
aff1Al[622, 0] := 1.11000E+04; aff1Al[622, 1] := 1.32983E-01;
aff1Al[623, 0] := 1.11500E+04; aff1Al[623, 1] := 1.32055E-01;
aff1Al[624, 0] := 1.12000E+04; aff1Al[624, 1] := 1.31136E-01;
aff1Al[625, 0] := 1.12500E+04; aff1Al[625, 1] := 1.30225E-01;
aff1Al[626, 0] := 1.13000E+04; aff1Al[626, 1] := 1.29321E-01;
aff1Al[627, 0] := 1.13500E+04; aff1Al[627, 1] := 1.28426E-01;
aff1Al[628, 0] := 1.14000E+04; aff1Al[628, 1] := 1.27538E-01;
aff1Al[629, 0] := 1.14500E+04; aff1Al[629, 1] := 1.26658E-01;
aff1Al[630, 0] := 1.15000E+04; aff1Al[630, 1] := 1.25786E-01;
aff1Al[631, 0] := 1.15500E+04; aff1Al[631, 1] := 1.24921E-01;
aff1Al[632, 0] := 1.16000E+04; aff1Al[632, 1] := 1.24065E-01;
aff1Al[633, 0] := 1.16500E+04; aff1Al[633, 1] := 1.23215E-01;
aff1Al[634, 0] := 1.17000E+04; aff1Al[634, 1] := 1.22373E-01;
aff1Al[635, 0] := 1.17500E+04; aff1Al[635, 1] := 1.21538E-01;
aff1Al[636, 0] := 1.18000E+04; aff1Al[636, 1] := 1.20711E-01;
aff1Al[637, 0] := 1.18500E+04; aff1Al[637, 1] := 1.19891E-01;
aff1Al[638, 0] := 1.19000E+04; aff1Al[638, 1] := 1.19078E-01;
aff1Al[639, 0] := 1.19500E+04; aff1Al[639, 1] := 1.18272E-01;
aff1Al[640, 0] := 1.20000E+04; aff1Al[640, 1] := 1.17473E-01;
aff1Al[641, 0] := 1.20500E+04; aff1Al[641, 1] := 1.16681E-01;
aff1Al[642, 0] := 1.21000E+04; aff1Al[642, 1] := 1.15896E-01;
aff1Al[643, 0] := 1.21500E+04; aff1Al[643, 1] := 1.15117E-01;
aff1Al[644, 0] := 1.22000E+04; aff1Al[644, 1] := 1.14346E-01;
aff1Al[645, 0] := 1.22500E+04; aff1Al[645, 1] := 1.13581E-01;
aff1Al[646, 0] := 1.23000E+04; aff1Al[646, 1] := 1.12823E-01;
aff1Al[647, 0] := 1.23500E+04; aff1Al[647, 1] := 1.12071E-01;
aff1Al[648, 0] := 1.24000E+04; aff1Al[648, 1] := 1.11326E-01;
aff1Al[649, 0] := 1.24500E+04; aff1Al[649, 1] := 1.10587E-01;
aff1Al[650, 0] := 1.25000E+04; aff1Al[650, 1] := 1.09854E-01;
aff1Al[651, 0] := 1.25500E+04; aff1Al[651, 1] := 1.09128E-01;
aff1Al[652, 0] := 1.26000E+04; aff1Al[652, 1] := 1.08408E-01;
aff1Al[653, 0] := 1.26500E+04; aff1Al[653, 1] := 1.07694E-01;
aff1Al[654, 0] := 1.27000E+04; aff1Al[654, 1] := 1.06986E-01;
aff1Al[655, 0] := 1.27500E+04; aff1Al[655, 1] := 1.06284E-01;
aff1Al[656, 0] := 1.28000E+04; aff1Al[656, 1] := 1.05588E-01;
aff1Al[657, 0] := 1.28500E+04; aff1Al[657, 1] := 1.04898E-01;
aff1Al[658, 0] := 1.29000E+04; aff1Al[658, 1] := 1.04214E-01;
aff1Al[659, 0] := 1.29500E+04; aff1Al[659, 1] := 1.03536E-01;
aff1Al[660, 0] := 1.30000E+04; aff1Al[660, 1] := 1.02863E-01;
aff1Al[661, 0] := 1.30500E+04; aff1Al[661, 1] := 1.02196E-01;
aff1Al[662, 0] := 1.31000E+04; aff1Al[662, 1] := 1.01535E-01;
aff1Al[663, 0] := 1.31500E+04; aff1Al[663, 1] := 1.00879E-01;
aff1Al[664, 0] := 1.32000E+04; aff1Al[664, 1] := 1.00229E-01;
aff1Al[665, 0] := 1.32500E+04; aff1Al[665, 1] := 9.95835E-02;
aff1Al[666, 0] := 1.33000E+04; aff1Al[666, 1] := 9.89440E-02;
aff1Al[667, 0] := 1.33500E+04; aff1Al[667, 1] := 9.83097E-02;
aff1Al[668, 0] := 1.34000E+04; aff1Al[668, 1] := 9.76807E-02;
aff1Al[669, 0] := 1.34500E+04; aff1Al[669, 1] := 9.70569E-02;
aff1Al[670, 0] := 1.35000E+04; aff1Al[670, 1] := 9.64382E-02;
aff1Al[671, 0] := 1.35500E+04; aff1Al[671, 1] := 9.58247E-02;
aff1Al[672, 0] := 1.36000E+04; aff1Al[672, 1] := 9.52161E-02;
aff1Al[673, 0] := 1.36500E+04; aff1Al[673, 1] := 9.46126E-02;
aff1Al[674, 0] := 1.37000E+04; aff1Al[674, 1] := 9.40140E-02;
aff1Al[675, 0] := 1.37500E+04; aff1Al[675, 1] := 9.34203E-02;
aff1Al[676, 0] := 1.38000E+04; aff1Al[676, 1] := 9.28314E-02;
aff1Al[677, 0] := 1.38500E+04; aff1Al[677, 1] := 9.22473E-02;
aff1Al[678, 0] := 1.39000E+04; aff1Al[678, 1] := 9.16680E-02;
aff1Al[679, 0] := 1.39500E+04; aff1Al[679, 1] := 9.10934E-02;
aff1Al[680, 0] := 1.40000E+04; aff1Al[680, 1] := 9.05234E-02;
aff1Al[681, 0] := 1.40500E+04; aff1Al[681, 1] := 8.99580E-02;
aff1Al[682, 0] := 1.41000E+04; aff1Al[682, 1] := 8.93971E-02;
aff1Al[683, 0] := 1.41500E+04; aff1Al[683, 1] := 8.88407E-02;
aff1Al[684, 0] := 1.42000E+04; aff1Al[684, 1] := 8.82888E-02;
aff1Al[685, 0] := 1.42500E+04; aff1Al[685, 1] := 8.77413E-02;
aff1Al[686, 0] := 1.43000E+04; aff1Al[686, 1] := 8.71981E-02;
aff1Al[687, 0] := 1.43500E+04; aff1Al[687, 1] := 8.66593E-02;
aff1Al[688, 0] := 1.44000E+04; aff1Al[688, 1] := 8.61247E-02;
aff1Al[689, 0] := 1.44500E+04; aff1Al[689, 1] := 8.55944E-02;
aff1Al[690, 0] := 1.45000E+04; aff1Al[690, 1] := 8.50682E-02;
aff1Al[691, 0] := 1.45500E+04; aff1Al[691, 1] := 8.45462E-02;
aff1Al[692, 0] := 1.46000E+04; aff1Al[692, 1] := 8.40283E-02;
aff1Al[693, 0] := 1.46500E+04; aff1Al[693, 1] := 8.35144E-02;
aff1Al[694, 0] := 1.47000E+04; aff1Al[694, 1] := 8.30046E-02;
aff1Al[695, 0] := 1.47500E+04; aff1Al[695, 1] := 8.24988E-02;
aff1Al[696, 0] := 1.48000E+04; aff1Al[696, 1] := 8.19969E-02;
aff1Al[697, 0] := 1.48500E+04; aff1Al[697, 1] := 8.14989E-02;
aff1Al[698, 0] := 1.49000E+04; aff1Al[698, 1] := 8.10047E-02;
aff1Al[699, 0] := 1.49500E+04; aff1Al[699, 1] := 8.05144E-02;
aff1Al[700, 0] := 1.50000E+04; aff1Al[700, 1] := 8.00278E-02;
aff1Al[701, 0] := 1.50500E+04; aff1Al[701, 1] := 7.95451E-02;
aff1Al[702, 0] := 1.51000E+04; aff1Al[702, 1] := 7.90660E-02;
aff1Al[703, 0] := 1.51500E+04; aff1Al[703, 1] := 7.85905E-02;
aff1Al[704, 0] := 1.52000E+04; aff1Al[704, 1] := 7.81187E-02;
aff1Al[705, 0] := 1.52500E+04; aff1Al[705, 1] := 7.76505E-02;
aff1Al[706, 0] := 1.53000E+04; aff1Al[706, 1] := 7.71859E-02;
aff1Al[707, 0] := 1.53500E+04; aff1Al[707, 1] := 7.67247E-02;
aff1Al[708, 0] := 1.54000E+04; aff1Al[708, 1] := 7.62671E-02;
aff1Al[709, 0] := 1.54500E+04; aff1Al[709, 1] := 7.58129E-02;
aff1Al[710, 0] := 1.55000E+04; aff1Al[710, 1] := 7.53622E-02;
aff1Al[711, 0] := 1.55500E+04; aff1Al[711, 1] := 7.49148E-02;
aff1Al[712, 0] := 1.56000E+04; aff1Al[712, 1] := 7.44708E-02;
aff1Al[713, 0] := 1.56500E+04; aff1Al[713, 1] := 7.40301E-02;
aff1Al[714, 0] := 1.57000E+04; aff1Al[714, 1] := 7.35927E-02;
aff1Al[715, 0] := 1.57500E+04; aff1Al[715, 1] := 7.31586E-02;
aff1Al[716, 0] := 1.58000E+04; aff1Al[716, 1] := 7.27277E-02;
aff1Al[717, 0] := 1.58500E+04; aff1Al[717, 1] := 7.23000E-02;
aff1Al[718, 0] := 1.59000E+04; aff1Al[718, 1] := 7.18755E-02;
aff1Al[719, 0] := 1.59500E+04; aff1Al[719, 1] := 7.14541E-02;
aff1Al[720, 0] := 1.60000E+04; aff1Al[720, 1] := 7.10357E-02;
aff1Al[721, 0] := 1.60500E+04; aff1Al[721, 1] := 7.06205E-02;
aff1Al[722, 0] := 1.61000E+04; aff1Al[722, 1] := 7.02083E-02;
aff1Al[723, 0] := 1.61500E+04; aff1Al[723, 1] := 6.97991E-02;
aff1Al[724, 0] := 1.62000E+04; aff1Al[724, 1] := 6.93929E-02;
aff1Al[725, 0] := 1.62500E+04; aff1Al[725, 1] := 6.89897E-02;
aff1Al[726, 0] := 1.63000E+04; aff1Al[726, 1] := 6.85894E-02;
aff1Al[727, 0] := 1.63500E+04; aff1Al[727, 1] := 6.81919E-02;
aff1Al[728, 0] := 1.64000E+04; aff1Al[728, 1] := 6.77974E-02;
aff1Al[729, 0] := 1.64500E+04; aff1Al[729, 1] := 6.74057E-02;
aff1Al[730, 0] := 1.65000E+04; aff1Al[730, 1] := 6.70168E-02;
aff1Al[731, 0] := 1.65500E+04; aff1Al[731, 1] := 6.66307E-02;
aff1Al[732, 0] := 1.66000E+04; aff1Al[732, 1] := 6.62474E-02;
aff1Al[733, 0] := 1.66500E+04; aff1Al[733, 1] := 6.58667E-02;
aff1Al[734, 0] := 1.67000E+04; aff1Al[734, 1] := 6.54888E-02;
aff1Al[735, 0] := 1.67500E+04; aff1Al[735, 1] := 6.51136E-02;
aff1Al[736, 0] := 1.68000E+04; aff1Al[736, 1] := 6.47411E-02;
aff1Al[737, 0] := 1.68500E+04; aff1Al[737, 1] := 6.43711E-02;
aff1Al[738, 0] := 1.69000E+04; aff1Al[738, 1] := 6.40038E-02;
aff1Al[739, 0] := 1.69500E+04; aff1Al[739, 1] := 6.36391E-02;
aff1Al[740, 0] := 1.70000E+04; aff1Al[740, 1] := 6.32770E-02;
aff1Al[741, 0] := 1.70500E+04; aff1Al[741, 1] := 6.29174E-02;
aff1Al[742, 0] := 1.71000E+04; aff1Al[742, 1] := 6.25603E-02;
aff1Al[743, 0] := 1.71500E+04; aff1Al[743, 1] := 6.22058E-02;
aff1Al[744, 0] := 1.72000E+04; aff1Al[744, 1] := 6.18536E-02;
aff1Al[745, 0] := 1.72500E+04; aff1Al[745, 1] := 6.15039E-02;
aff1Al[746, 0] := 1.73000E+04; aff1Al[746, 1] := 6.11566E-02;
aff1Al[747, 0] := 1.73500E+04; aff1Al[747, 1] := 6.08118E-02;
aff1Al[748, 0] := 1.74000E+04; aff1Al[748, 1] := 6.04693E-02;
aff1Al[749, 0] := 1.74500E+04; aff1Al[749, 1] := 6.01292E-02;
aff1Al[750, 0] := 1.75000E+04; aff1Al[750, 1] := 5.97915E-02;
aff1Al[751, 0] := 1.75500E+04; aff1Al[751, 1] := 5.94560E-02;
aff1Al[752, 0] := 1.76000E+04; aff1Al[752, 1] := 5.91228E-02;
aff1Al[753, 0] := 1.76500E+04; aff1Al[753, 1] := 5.87919E-02;
aff1Al[754, 0] := 1.77000E+04; aff1Al[754, 1] := 5.84633E-02;
aff1Al[755, 0] := 1.77500E+04; aff1Al[755, 1] := 5.81368E-02;
aff1Al[756, 0] := 1.78000E+04; aff1Al[756, 1] := 5.78126E-02;
aff1Al[757, 0] := 1.78500E+04; aff1Al[757, 1] := 5.74906E-02;
aff1Al[758, 0] := 1.79000E+04; aff1Al[758, 1] := 5.71707E-02;
aff1Al[759, 0] := 1.79500E+04; aff1Al[759, 1] := 5.68531E-02;
aff1Al[760, 0] := 1.80000E+04; aff1Al[760, 1] := 5.65375E-02;
aff1Al[761, 0] := 1.80500E+04; aff1Al[761, 1] := 5.62241E-02;
aff1Al[762, 0] := 1.81000E+04; aff1Al[762, 1] := 5.59127E-02;
aff1Al[763, 0] := 1.81500E+04; aff1Al[763, 1] := 5.56034E-02;
aff1Al[764, 0] := 1.82000E+04; aff1Al[764, 1] := 5.52962E-02;
aff1Al[765, 0] := 1.82500E+04; aff1Al[765, 1] := 5.49910E-02;
aff1Al[766, 0] := 1.83000E+04; aff1Al[766, 1] := 5.46879E-02;
aff1Al[767, 0] := 1.83500E+04; aff1Al[767, 1] := 5.43868E-02;
aff1Al[768, 0] := 1.84000E+04; aff1Al[768, 1] := 5.40876E-02;
aff1Al[769, 0] := 1.84500E+04; aff1Al[769, 1] := 5.37905E-02;
aff1Al[770, 0] := 1.85000E+04; aff1Al[770, 1] := 5.34953E-02;
aff1Al[771, 0] := 1.85500E+04; aff1Al[771, 1] := 5.32020E-02;
aff1Al[772, 0] := 1.86000E+04; aff1Al[772, 1] := 5.29106E-02;
aff1Al[773, 0] := 1.86500E+04; aff1Al[773, 1] := 5.26211E-02;
aff1Al[774, 0] := 1.87000E+04; aff1Al[774, 1] := 5.23335E-02;
aff1Al[775, 0] := 1.87500E+04; aff1Al[775, 1] := 5.20478E-02;
aff1Al[776, 0] := 1.88000E+04; aff1Al[776, 1] := 5.17639E-02;
aff1Al[777, 0] := 1.88500E+04; aff1Al[777, 1] := 5.14818E-02;
aff1Al[778, 0] := 1.89000E+04; aff1Al[778, 1] := 5.12016E-02;
aff1Al[779, 0] := 1.89500E+04; aff1Al[779, 1] := 5.09232E-02;
aff1Al[780, 0] := 1.90000E+04; aff1Al[780, 1] := 5.06466E-02;
aff1Al[781, 0] := 1.90500E+04; aff1Al[781, 1] := 5.03717E-02;
aff1Al[782, 0] := 1.91000E+04; aff1Al[782, 1] := 5.00986E-02;
aff1Al[783, 0] := 1.91500E+04; aff1Al[783, 1] := 4.98273E-02;
aff1Al[784, 0] := 1.92000E+04; aff1Al[784, 1] := 4.95577E-02;
aff1Al[785, 0] := 1.92500E+04; aff1Al[785, 1] := 4.92898E-02;
aff1Al[786, 0] := 1.93000E+04; aff1Al[786, 1] := 4.90236E-02;
aff1Al[787, 0] := 1.93500E+04; aff1Al[787, 1] := 4.87591E-02;
aff1Al[788, 0] := 1.94000E+04; aff1Al[788, 1] := 4.84962E-02;
aff1Al[789, 0] := 1.94500E+04; aff1Al[789, 1] := 4.82350E-02;
aff1Al[790, 0] := 1.95000E+04; aff1Al[790, 1] := 4.79755E-02;
aff1Al[791, 0] := 1.95500E+04; aff1Al[791, 1] := 4.77175E-02;
aff1Al[792, 0] := 1.96000E+04; aff1Al[792, 1] := 4.74612E-02;
aff1Al[793, 0] := 1.96500E+04; aff1Al[793, 1] := 4.72066E-02;
aff1Al[794, 0] := 1.97000E+04; aff1Al[794, 1] := 4.69535E-02;
aff1Al[795, 0] := 1.97500E+04; aff1Al[795, 1] := 4.67019E-02;
aff1Al[796, 0] := 1.98000E+04; aff1Al[796, 1] := 4.64520E-02;
aff1Al[797, 0] := 1.98500E+04; aff1Al[797, 1] := 4.62035E-02;
aff1Al[798, 0] := 1.99000E+04; aff1Al[798, 1] := 4.59566E-02;
aff1Al[799, 0] := 1.99500E+04; aff1Al[799, 1] := 4.57112E-02;
aff1Al[800, 0] := 2.00000E+04; aff1Al[800, 1] := 4.54674E-02;
aff1Al[801, 0] := 2.00500E+04; aff1Al[801, 1] := 4.52250E-02;
aff1Al[802, 0] := 2.01000E+04; aff1Al[802, 1] := 4.49841E-02;
aff1Al[803, 0] := 2.01500E+04; aff1Al[803, 1] := 4.47447E-02;
aff1Al[804, 0] := 2.02000E+04; aff1Al[804, 1] := 4.45068E-02;
aff1Al[805, 0] := 2.02500E+04; aff1Al[805, 1] := 4.42704E-02;
aff1Al[806, 0] := 2.03000E+04; aff1Al[806, 1] := 4.40353E-02;
aff1Al[807, 0] := 2.03500E+04; aff1Al[807, 1] := 4.38017E-02;
aff1Al[808, 0] := 2.04000E+04; aff1Al[808, 1] := 4.35695E-02;
aff1Al[809, 0] := 2.04500E+04; aff1Al[809, 1] := 4.33387E-02;
aff1Al[810, 0] := 2.05000E+04; aff1Al[810, 1] := 4.31093E-02;
aff1Al[811, 0] := 2.05500E+04; aff1Al[811, 1] := 4.28812E-02;
aff1Al[812, 0] := 2.06000E+04; aff1Al[812, 1] := 4.26546E-02;
aff1Al[813, 0] := 2.06500E+04; aff1Al[813, 1] := 4.24293E-02;
aff1Al[814, 0] := 2.07000E+04; aff1Al[814, 1] := 4.22053E-02;
aff1Al[815, 0] := 2.07500E+04; aff1Al[815, 1] := 4.19827E-02;
aff1Al[816, 0] := 2.08000E+04; aff1Al[816, 1] := 4.17614E-02;
aff1Al[817, 0] := 2.08500E+04; aff1Al[817, 1] := 4.15415E-02;
aff1Al[818, 0] := 2.09000E+04; aff1Al[818, 1] := 4.13228E-02;
aff1Al[819, 0] := 2.09500E+04; aff1Al[819, 1] := 4.11054E-02;
aff1Al[820, 0] := 2.10000E+04; aff1Al[820, 1] := 4.08893E-02;
aff1Al[821, 0] := 2.10500E+04; aff1Al[821, 1] := 4.06745E-02;
aff1Al[822, 0] := 2.11000E+04; aff1Al[822, 1] := 4.04609E-02;
aff1Al[823, 0] := 2.11500E+04; aff1Al[823, 1] := 4.02486E-02;
aff1Al[824, 0] := 2.12000E+04; aff1Al[824, 1] := 4.00376E-02;
aff1Al[825, 0] := 2.12500E+04; aff1Al[825, 1] := 3.98278E-02;
aff1Al[826, 0] := 2.13000E+04; aff1Al[826, 1] := 3.96192E-02;
aff1Al[827, 0] := 2.13500E+04; aff1Al[827, 1] := 3.94118E-02;
aff1Al[828, 0] := 2.14000E+04; aff1Al[828, 1] := 3.92056E-02;
aff1Al[829, 0] := 2.14500E+04; aff1Al[829, 1] := 3.90007E-02;
aff1Al[830, 0] := 2.15000E+04; aff1Al[830, 1] := 3.87969E-02;
aff1Al[831, 0] := 2.15500E+04; aff1Al[831, 1] := 3.85944E-02;
aff1Al[832, 0] := 2.16000E+04; aff1Al[832, 1] := 3.83929E-02;
aff1Al[833, 0] := 2.16500E+04; aff1Al[833, 1] := 3.81927E-02;
aff1Al[834, 0] := 2.17000E+04; aff1Al[834, 1] := 3.79935E-02;
aff1Al[835, 0] := 2.17500E+04; aff1Al[835, 1] := 3.77955E-02;
aff1Al[836, 0] := 2.18000E+04; aff1Al[836, 1] := 3.75986E-02;
aff1Al[837, 0] := 2.18500E+04; aff1Al[837, 1] := 3.74029E-02;
aff1Al[838, 0] := 2.19000E+04; aff1Al[838, 1] := 3.72083E-02;
aff1Al[839, 0] := 2.19500E+04; aff1Al[839, 1] := 3.70148E-02;
aff1Al[840, 0] := 2.20000E+04; aff1Al[840, 1] := 3.68225E-02;
aff1Al[841, 0] := 2.20500E+04; aff1Al[841, 1] := 3.66311E-02;
aff1Al[842, 0] := 2.21000E+04; aff1Al[842, 1] := 3.64409E-02;
aff1Al[843, 0] := 2.21500E+04; aff1Al[843, 1] := 3.62517E-02;
aff1Al[844, 0] := 2.22000E+04; aff1Al[844, 1] := 3.60636E-02;
aff1Al[845, 0] := 2.22500E+04; aff1Al[845, 1] := 3.58766E-02;
aff1Al[846, 0] := 2.23000E+04; aff1Al[846, 1] := 3.56906E-02;
aff1Al[847, 0] := 2.23500E+04; aff1Al[847, 1] := 3.55057E-02;
aff1Al[848, 0] := 2.24000E+04; aff1Al[848, 1] := 3.53218E-02;
aff1Al[849, 0] := 2.24500E+04; aff1Al[849, 1] := 3.51389E-02;
aff1Al[850, 0] := 2.25000E+04; aff1Al[850, 1] := 3.49571E-02;
aff1Al[851, 0] := 2.25500E+04; aff1Al[851, 1] := 3.47762E-02;
aff1Al[852, 0] := 2.26000E+04; aff1Al[852, 1] := 3.45963E-02;
aff1Al[853, 0] := 2.26500E+04; aff1Al[853, 1] := 3.44175E-02;
aff1Al[854, 0] := 2.27000E+04; aff1Al[854, 1] := 3.42396E-02;
aff1Al[855, 0] := 2.27500E+04; aff1Al[855, 1] := 3.40627E-02;
aff1Al[856, 0] := 2.28000E+04; aff1Al[856, 1] := 3.38869E-02;
aff1Al[857, 0] := 2.28500E+04; aff1Al[857, 1] := 3.37119E-02;
aff1Al[858, 0] := 2.29000E+04; aff1Al[858, 1] := 3.35380E-02;
aff1Al[859, 0] := 2.29500E+04; aff1Al[859, 1] := 3.33650E-02;
aff1Al[860, 0] := 2.30000E+04; aff1Al[860, 1] := 3.31929E-02;
aff1Al[861, 0] := 2.30500E+04; aff1Al[861, 1] := 3.30217E-02;
aff1Al[862, 0] := 2.31000E+04; aff1Al[862, 1] := 3.28515E-02;
aff1Al[863, 0] := 2.31500E+04; aff1Al[863, 1] := 3.26822E-02;
aff1Al[864, 0] := 2.32000E+04; aff1Al[864, 1] := 3.25139E-02;
aff1Al[865, 0] := 2.32500E+04; aff1Al[865, 1] := 3.23464E-02;
aff1Al[866, 0] := 2.33000E+04; aff1Al[866, 1] := 3.21799E-02;
aff1Al[867, 0] := 2.33500E+04; aff1Al[867, 1] := 3.20142E-02;
aff1Al[868, 0] := 2.34000E+04; aff1Al[868, 1] := 3.18495E-02;
aff1Al[869, 0] := 2.34500E+04; aff1Al[869, 1] := 3.16856E-02;
aff1Al[870, 0] := 2.35000E+04; aff1Al[870, 1] := 3.15226E-02;
aff1Al[871, 0] := 2.35500E+04; aff1Al[871, 1] := 3.13605E-02;
aff1Al[872, 0] := 2.36000E+04; aff1Al[872, 1] := 3.11993E-02;
aff1Al[873, 0] := 2.36500E+04; aff1Al[873, 1] := 3.10389E-02;
aff1Al[874, 0] := 2.37000E+04; aff1Al[874, 1] := 3.08793E-02;
aff1Al[875, 0] := 2.37500E+04; aff1Al[875, 1] := 3.07206E-02;
aff1Al[876, 0] := 2.38000E+04; aff1Al[876, 1] := 3.05628E-02;
aff1Al[877, 0] := 2.38500E+04; aff1Al[877, 1] := 3.04058E-02;
aff1Al[878, 0] := 2.39000E+04; aff1Al[878, 1] := 3.02496E-02;
aff1Al[879, 0] := 2.39500E+04; aff1Al[879, 1] := 3.00943E-02;
aff1Al[880, 0] := 2.40000E+04; aff1Al[880, 1] := 2.99397E-02;
aff1Al[881, 0] := 2.40500E+04; aff1Al[881, 1] := 2.97860E-02;
aff1Al[882, 0] := 2.41000E+04; aff1Al[882, 1] := 2.96331E-02;
aff1Al[883, 0] := 2.41500E+04; aff1Al[883, 1] := 2.94810E-02;
aff1Al[884, 0] := 2.42000E+04; aff1Al[884, 1] := 2.93297E-02;
aff1Al[885, 0] := 2.42500E+04; aff1Al[885, 1] := 2.91791E-02;
aff1Al[886, 0] := 2.43000E+04; aff1Al[886, 1] := 2.90294E-02;
aff1Al[887, 0] := 2.43500E+04; aff1Al[887, 1] := 2.88804E-02;
aff1Al[888, 0] := 2.44000E+04; aff1Al[888, 1] := 2.87323E-02;
aff1Al[889, 0] := 2.44500E+04; aff1Al[889, 1] := 2.85849E-02;
aff1Al[890, 0] := 2.45000E+04; aff1Al[890, 1] := 2.84382E-02;
aff1Al[891, 0] := 2.45500E+04; aff1Al[891, 1] := 2.82923E-02;
aff1Al[892, 0] := 2.46000E+04; aff1Al[892, 1] := 2.81472E-02;
aff1Al[893, 0] := 2.46500E+04; aff1Al[893, 1] := 2.80028E-02;
aff1Al[894, 0] := 2.47000E+04; aff1Al[894, 1] := 2.78591E-02;
aff1Al[895, 0] := 2.47500E+04; aff1Al[895, 1] := 2.77162E-02;
aff1Al[896, 0] := 2.48000E+04; aff1Al[896, 1] := 2.75740E-02;
aff1Al[897, 0] := 2.48500E+04; aff1Al[897, 1] := 2.74326E-02;
aff1Al[898, 0] := 2.49000E+04; aff1Al[898, 1] := 2.72918E-02;
aff1Al[899, 0] := 2.49500E+04; aff1Al[899, 1] := 2.71518E-02;
aff1Al[900, 0] := 2.50000E+04; aff1Al[900, 1] := 2.70125E-02;
aff1Al[901, 0] := 2.50500E+04; aff1Al[901, 1] := 2.68738E-02;
aff1Al[902, 0] := 2.51000E+04; aff1Al[902, 1] := 2.67359E-02;
aff1Al[903, 0] := 2.51500E+04; aff1Al[903, 1] := 2.65987E-02;
aff1Al[904, 0] := 2.52000E+04; aff1Al[904, 1] := 2.64622E-02;
aff1Al[905, 0] := 2.52500E+04; aff1Al[905, 1] := 2.63264E-02;
aff1Al[906, 0] := 2.53000E+04; aff1Al[906, 1] := 2.61913E-02;
aff1Al[907, 0] := 2.53500E+04; aff1Al[907, 1] := 2.60568E-02;
aff1Al[908, 0] := 2.54000E+04; aff1Al[908, 1] := 2.59230E-02;
aff1Al[909, 0] := 2.54500E+04; aff1Al[909, 1] := 2.57899E-02;
aff1Al[910, 0] := 2.55000E+04; aff1Al[910, 1] := 2.56575E-02;
aff1Al[911, 0] := 2.55500E+04; aff1Al[911, 1] := 2.55257E-02;
aff1Al[912, 0] := 2.56000E+04; aff1Al[912, 1] := 2.53946E-02;
aff1Al[913, 0] := 2.56500E+04; aff1Al[913, 1] := 2.52641E-02;
aff1Al[914, 0] := 2.57000E+04; aff1Al[914, 1] := 2.51342E-02;
aff1Al[915, 0] := 2.57500E+04; aff1Al[915, 1] := 2.50051E-02;
aff1Al[916, 0] := 2.58000E+04; aff1Al[916, 1] := 2.48765E-02;
aff1Al[917, 0] := 2.58500E+04; aff1Al[917, 1] := 2.47486E-02;
aff1Al[918, 0] := 2.59000E+04; aff1Al[918, 1] := 2.46213E-02;
aff1Al[919, 0] := 2.59500E+04; aff1Al[919, 1] := 2.44947E-02;
aff1Al[920, 0] := 2.60000E+04; aff1Al[920, 1] := 2.43687E-02;
aff1Al[921, 0] := 2.60500E+04; aff1Al[921, 1] := 2.42433E-02;
aff1Al[922, 0] := 2.61000E+04; aff1Al[922, 1] := 2.41185E-02;
aff1Al[923, 0] := 2.61500E+04; aff1Al[923, 1] := 2.39945E-02;
aff1Al[924, 0] := 2.62000E+04; aff1Al[924, 1] := 2.38710E-02;
aff1Al[925, 0] := 2.62500E+04; aff1Al[925, 1] := 2.37481E-02;
aff1Al[926, 0] := 2.63000E+04; aff1Al[926, 1] := 2.36256E-02;
aff1Al[927, 0] := 2.63500E+04; aff1Al[927, 1] := 2.35035E-02;
aff1Al[928, 0] := 2.64000E+04; aff1Al[928, 1] := 2.33814E-02;
aff1Al[929, 0] := 2.64500E+04; aff1Al[929, 1] := 2.32598E-02;
aff1Al[930, 0] := 2.65000E+04; aff1Al[930, 1] := 2.31392E-02;
aff1Al[931, 0] := 2.65500E+04; aff1Al[931, 1] := 2.30200E-02;
aff1Al[932, 0] := 2.66000E+04; aff1Al[932, 1] := 2.29027E-02;
aff1Al[933, 0] := 2.66500E+04; aff1Al[933, 1] := 2.27879E-02;
aff1Al[934, 0] := 2.67000E+04; aff1Al[934, 1] := 2.26752E-02;
aff1Al[935, 0] := 2.67500E+04; aff1Al[935, 1] := 2.25643E-02;
aff1Al[936, 0] := 2.68000E+04; aff1Al[936, 1] := 2.24548E-02;
aff1Al[937, 0] := 2.68500E+04; aff1Al[937, 1] := 2.23461E-02;
aff1Al[938, 0] := 2.69000E+04; aff1Al[938, 1] := 2.22378E-02;
aff1Al[939, 0] := 2.69500E+04; aff1Al[939, 1] := 2.21298E-02;
aff1Al[940, 0] := 2.70000E+04; aff1Al[940, 1] := 2.20219E-02;
aff1Al[941, 0] := 2.70500E+04; aff1Al[941, 1] := 2.19142E-02;
aff1Al[942, 0] := 2.71000E+04; aff1Al[942, 1] := 2.18067E-02;
aff1Al[943, 0] := 2.71500E+04; aff1Al[943, 1] := 2.16993E-02;
aff1Al[944, 0] := 2.72000E+04; aff1Al[944, 1] := 2.15921E-02;
aff1Al[945, 0] := 2.72500E+04; aff1Al[945, 1] := 2.14851E-02;
aff1Al[946, 0] := 2.73000E+04; aff1Al[946, 1] := 2.13782E-02;
aff1Al[947, 0] := 2.73500E+04; aff1Al[947, 1] := 2.12715E-02;
aff1Al[948, 0] := 2.74000E+04; aff1Al[948, 1] := 2.11651E-02;
aff1Al[949, 0] := 2.74500E+04; aff1Al[949, 1] := 2.10590E-02;
aff1Al[950, 0] := 2.75000E+04; aff1Al[950, 1] := 2.09532E-02;
aff1Al[951, 0] := 2.75500E+04; aff1Al[951, 1] := 2.08477E-02;
aff1Al[952, 0] := 2.76000E+04; aff1Al[952, 1] := 2.07426E-02;
aff1Al[953, 0] := 2.76500E+04; aff1Al[953, 1] := 2.06379E-02;
aff1Al[954, 0] := 2.77000E+04; aff1Al[954, 1] := 2.05334E-02;
aff1Al[955, 0] := 2.77500E+04; aff1Al[955, 1] := 2.04293E-02;
aff1Al[956, 0] := 2.78000E+04; aff1Al[956, 1] := 2.03256E-02;
aff1Al[957, 0] := 2.78500E+04; aff1Al[957, 1] := 2.02222E-02;
aff1Al[958, 0] := 2.79000E+04; aff1Al[958, 1] := 2.01192E-02;
aff1Al[959, 0] := 2.79500E+04; aff1Al[959, 1] := 2.00166E-02;
aff1Al[960, 0] := 2.80000E+04; aff1Al[960, 1] := 1.99143E-02;
aff1Al[961, 0] := 2.80500E+04; aff1Al[961, 1] := 1.98124E-02;
aff1Al[962, 0] := 2.81000E+04; aff1Al[962, 1] := 1.97108E-02;
aff1Al[963, 0] := 2.81500E+04; aff1Al[963, 1] := 1.96096E-02;
aff1Al[964, 0] := 2.82000E+04; aff1Al[964, 1] := 1.95088E-02;
aff1Al[965, 0] := 2.82500E+04; aff1Al[965, 1] := 1.94084E-02;
aff1Al[966, 0] := 2.83000E+04; aff1Al[966, 1] := 1.93083E-02;
aff1Al[967, 0] := 2.83500E+04; aff1Al[967, 1] := 1.92087E-02;
aff1Al[968, 0] := 2.84000E+04; aff1Al[968, 1] := 1.91094E-02;
aff1Al[969, 0] := 2.84500E+04; aff1Al[969, 1] := 1.90104E-02;
aff1Al[970, 0] := 2.85000E+04; aff1Al[970, 1] := 1.89119E-02;
aff1Al[971, 0] := 2.85500E+04; aff1Al[971, 1] := 1.88137E-02;
aff1Al[972, 0] := 2.86000E+04; aff1Al[972, 1] := 1.87159E-02;
aff1Al[973, 0] := 2.86500E+04; aff1Al[973, 1] := 1.86185E-02;
aff1Al[974, 0] := 2.87000E+04; aff1Al[974, 1] := 1.85215E-02;
aff1Al[975, 0] := 2.87500E+04; aff1Al[975, 1] := 1.84248E-02;
aff1Al[976, 0] := 2.88000E+04; aff1Al[976, 1] := 1.83286E-02;
aff1Al[977, 0] := 2.88500E+04; aff1Al[977, 1] := 1.82327E-02;
aff1Al[978, 0] := 2.89000E+04; aff1Al[978, 1] := 1.81371E-02;
aff1Al[979, 0] := 2.89500E+04; aff1Al[979, 1] := 1.80420E-02;
aff1Al[980, 0] := 2.90000E+04; aff1Al[980, 1] := 1.79472E-02;
aff1Al[981, 0] := 2.90500E+04; aff1Al[981, 1] := 1.78528E-02;
aff1Al[982, 0] := 2.91000E+04; aff1Al[982, 1] := 1.77588E-02;
aff1Al[983, 0] := 2.91500E+04; aff1Al[983, 1] := 1.76652E-02;
aff1Al[984, 0] := 2.92000E+04; aff1Al[984, 1] := 1.75719E-02;
aff1Al[985, 0] := 2.92500E+04; aff1Al[985, 1] := 1.74790E-02;
aff1Al[986, 0] := 2.93000E+04; aff1Al[986, 1] := 1.73864E-02;
aff1Al[987, 0] := 2.93500E+04; aff1Al[987, 1] := 1.72943E-02;
aff1Al[988, 0] := 2.94000E+04; aff1Al[988, 1] := 1.72025E-02;
aff1Al[989, 0] := 2.94500E+04; aff1Al[989, 1] := 1.71110E-02;
aff1Al[990, 0] := 2.95000E+04; aff1Al[990, 1] := 1.70199E-02;
aff1Al[991, 0] := 2.95500E+04; aff1Al[991, 1] := 1.69292E-02;
aff1Al[992, 0] := 2.96000E+04; aff1Al[992, 1] := 1.68389E-02;
aff1Al[993, 0] := 2.96500E+04; aff1Al[993, 1] := 1.67489E-02;
aff1Al[994, 0] := 2.97000E+04; aff1Al[994, 1] := 1.66592E-02;
aff1Al[995, 0] := 2.97500E+04; aff1Al[995, 1] := 1.65699E-02;
aff1Al[996, 0] := 2.98000E+04; aff1Al[996, 1] := 1.64810E-02;
aff1Al[997, 0] := 2.98500E+04; aff1Al[997, 1] := 1.63925E-02;
aff1Al[998, 0] := 2.99000E+04; aff1Al[998, 1] := 1.63043E-02;
aff1Al[999, 0] := 2.99500E+04; aff1Al[999, 1] := 1.62164E-02;

// Element = Si

